// TIA Portal V20 export
// export: Created 2025-12-01T14:57:41.7461211Z, ExportSetting None, DisplayName Totally Integrated Automation Portal, DisplayVersion V20 Update 3, DisplayName TIA Portal Openness, DisplayVersion V20 Update 3, DisplayName TIA Portal Version Control Interface, DisplayVersion V20 Update 3, DisplayName STEP 7 Professional, DisplayVersion V20 Update 3, DisplayName STEP 7 Safety, DisplayVersion V20 Update 2, DisplayName WinCC Basic/Comfort/Advanced, DisplayVersion V20 Update 3, DisplayName WinCC Professional, DisplayVersion V20 Update 3, DisplayName WinCC Unified, DisplayVersion V20 Update 3
FUNCTION_BLOCK "FB381_Transporte_Paletizador_NDD_E12_S23"   // FB381, LAD
TITLE = Control del Ramal de Salidas
{ S7_Optimized_Access := 'FALSE' }
AUTHOR : PASO
NAME : 20160509
VERSION : 3.6
// E1E3_S1S3    (Paletizador NDD)
// stored: AutoNumber false, SetENOAutomatically false
   VAR_INPUT
      Mesa : UInt;   // Mesa de la FB
      Error_Tx : Bool;
      EnTension : Bool;   // Existe Tension en la Mesa
      Termico_Tx : Bool;
      pHsMx_1 : Bool;   // Desactiva si Transferencia controlada
      pHsMx_2 : Bool;   // Desactiva si Transferencia controlada
      pHsMx_PR1 : Bool;   // Si no hay Prot ON
      pHsMx_PR3 : Bool;   // Si no hay Prot ON
      pHsMx_CorteVelo : Bool;
      phsMx_Seguridad : Bool;
      Avance_Tx : Bool;
      Retroceso_Tx : Bool;
      MAnt_DescargaAct_M1 : Bool;
      AVTF_Ent_M1 : Bool;
      P_Mens_Ent_M1 : Bool;
      MAnt_DescargaAct_M3 : Bool;
      AVTF_Ent_M3 : Bool;
      P_Mens_Ent_M3 : Bool;
      PTF_Sal_M1 : Bool;
      FTF_Sal_M1 : Bool;
      PTF_Sal_M3 : Bool;
      FTF_Sal_M3 : Bool;
      Mx_VelocidadLenta_In : Bool;   // Forzar a Velociada Lenta
      F_EnvMens_Mx : Bool;
      OrdSal_S01 : Bool;
      OrdSal_S03 : Bool;
      V_CNT_pHsMx : Int := 300;
      V_CNT_pHsMx_FTF : Int := 50;   // Valor contador para FTF_Mant
      V_CNTSeg_pHsMx : Int := 3000;
      V_CNT_PasoLenta : Int := 3000;
      V_CNT_ApHsMx : Int := 500;
      V_CNTSeg_ApHsMx : Int := 3000;
      V_CNT_pHsMx_E0S0 : Int := 2000;
      V_CNT_Simultaneo : Int := 2000;
      V_InicioSimultaneo : Int := 0;
      V_FinSimultaneo : Int := 0;
      V_TOut_Tx_Mx : Int := 30000;
      V_TMP_Protrusion : Int := 500;
      V_CNT_PerdidapHs : Int := 1000;
   END_VAR
   VAR_OUTPUT
      P_EnvMens_PMx : Bool;
      P_RecepOK_Mx : Bool;
      PTF_Ent_M1 : Bool;
      FTF_Ent_M1 : Bool;
      PTF_Ent_M3 : Bool;
      FTF_Ent_M3 : Bool;
      ATF_Sal_M1 : Bool;
      P_Mens_Sal_M1 : Bool;
      ATF_Sal_M3 : Bool;
      P_Mens_Sal_M3 : Bool;
   END_VAR
   VAR_IN_OUT
      Interlock_TELEV : "NDD_Interlock_TElev";
   END_VAR
   VAR
      Anular_prE1 : Bool;   // ???
      Anular_prS3 : Bool;   // ???
      Mx_ET00 : Bool;
      Mx_ET01 : Bool;
      Mx_ET02 : Bool;
      Mx_ET08 : Bool;
      Mx_ET09 : Bool;
      Mx_ET10 : Bool;
      Mx_ET11 : Bool;
      Mx_ET12 : Bool;
      Mx_ET50 : Bool;
      Mx_ET51 : Bool;
      Mx_ET110 : Bool;
      Mx_ET111 : Bool;
      Mx_ET150 : Bool;
      Mx_ET151 : Bool;
      Mx_ET30 : Bool;
      Mx_ET31 : Bool;
      Mx_ET32 : Bool;
      Mx_ET33 : Bool;
      Mx_ET70 : Bool;
      Mx_ET71 : Bool;
      Mx_ET72 : Bool;
      Selec_M1_Entrada : Bool;
      Selec_M3_Entrada : Bool;
      Selec_M0_Entrada : Bool;
      Selec_M1_Salida : Bool;
      Selec_M3_Salida : Bool;
      Select_M0_Salida : Bool;
      MEnt_DescargaAct : Bool;
      AVTF_MEnt : Bool;
      P_Mens_MEnt : Bool;
      PTF_MEnt : Bool;
      FTF_MEnt : Bool;
      AVTF_MSal : Bool;
      P_Mens_MSal : Bool;
      PTF_MSal : Bool;
      FTF_MSal : Bool;
      FTF_MEnt_M0 : Bool;
      ProtocoloIniciado : Bool;
      CNT_pHsMx_FTF_OK : Bool;
      Simultaneo_Mx : Bool;
      CNT_pHsMx { S7_SetPoint := 'True'} : "FB910_CNT_UHS";
      CNTSeg_pHsMx { S7_SetPoint := 'True'} : "FB910_CNT_UHS";
      CNT_ApHsMx { S7_SetPoint := 'True'} : "FB910_CNT_UHS";
      CNTSeg_ApHsMx { S7_SetPoint := 'True'} : "FB910_CNT_UHS";
      CNT_Simultaneo { S7_SetPoint := 'True'} : "FB910_CNT_UHS";
      CNTEntrada_E0 { S7_SetPoint := 'True'} : "FB910_CNT_UHS";
      CNTSalida_S0 { S7_SetPoint := 'True'} : "FB910_CNT_UHS";
      TMP_EnTension { S7_SetPoint := 'True'} : "FB910_CNT_UHS";
      TOut_Av_Mx { S7_SetPoint := 'True'} : "FB910_CNT_UHS";
      TOut_Ret_Mx { S7_SetPoint := 'True'} : "FB910_CNT_UHS";
      TMP_Protrusion { S7_SetPoint := 'True'} : "FB910_CNT_UHS";
      CNT_PerdidapHs { S7_SetPoint := 'True'} : "FB910_CNT_UHS";
      STAT_EnvMens_PMx : Bool;
   END_VAR
   VAR_TEMP
      EstadoZona : "EstadoZona";
      EstadoVI : "EstadosMesa_Transporte_Paletizador_NDD";
      ConfigFB : "UDT_ConfigFB";   // Configuracion de la FB de la Mesa
      V_Protrusion : Int;
      Aux_ET00 : Bool;
      SinPHS_E0 : Bool;
   END_VAR
   VAR_TEMP   // added for the SCL form of the ladder/FBD networks
      _w1 : Bool;
      _w2 : Bool;
   END_VAR
BEGIN

REGION Network 1: INICIALIZACIONES
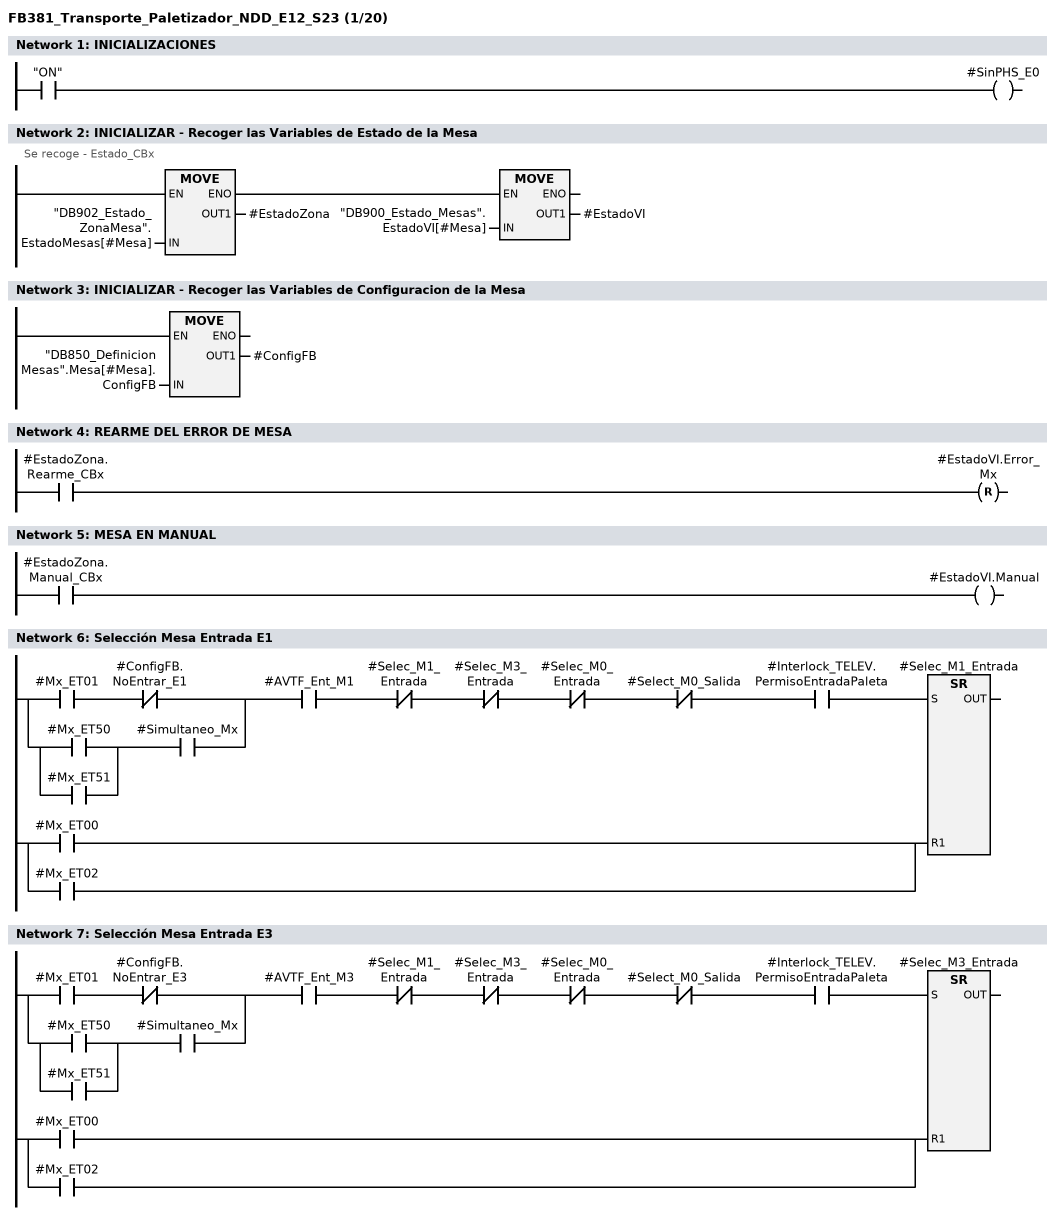
   RUNG wire#powerrail
      Contact( "ON" )
      Coil( #SinPHS_E0 )
   END_RUNG
   // the same network as SCL:
   #SinPHS_E0 := "ON";
END_REGION

REGION Network 2: INICIALIZAR - Recoger las Variables de Estado de la Mesa
   // Se recoge - Estado_CBx
   RUNG wire#powerrail
      Move(in := "DB902_Estado_ZonaMesa".EstadoMesas[#Mesa], out1 => #EstadoZona)
      Move(in := "DB900_Estado_Mesas".EstadoVI[#Mesa], out1 => #EstadoVI)
   END_RUNG
   // the same network as SCL:
   #EstadoZona := "DB902_Estado_ZonaMesa".EstadoMesas[#Mesa];
   #EstadoVI := "DB900_Estado_Mesas".EstadoVI[#Mesa];
END_REGION

REGION Network 3: INICIALIZAR - Recoger las Variables de Configuracion de la Mesa
   RUNG wire#powerrail
      Move(in := "DB850_DefinicionMesas".Mesa[#Mesa].ConfigFB, out1 => #ConfigFB)
   END_RUNG
   // the same network as SCL:
   #ConfigFB := "DB850_DefinicionMesas".Mesa[#Mesa].ConfigFB;
END_REGION

REGION Network 4: REARME DEL ERROR DE MESA
   RUNG wire#powerrail
      Contact( #EstadoZona.Rearme_CBx )
      R_Coil( #EstadoVI.Error_Mx )
   END_RUNG
   // the same network as SCL:
   IF #EstadoZona.Rearme_CBx THEN #EstadoVI.Error_Mx := FALSE; END_IF;
END_REGION

REGION Network 5: MESA EN MANUAL
   RUNG wire#powerrail
      Contact( #EstadoZona.Manual_CBx )
      Coil( #EstadoVI.Manual )
   END_RUNG
   // the same network as SCL:
   #EstadoVI.Manual := #EstadoZona.Manual_CBx;
END_REGION

REGION Network 6: Selección Mesa Entrada E1
   RUNG wire#powerrail
      Contact( #Mx_ET01 )
      I_Contact( #ConfigFB.NoEntrar_E1 )
      wire#w1
      Contact( #AVTF_Ent_M1 )
      I_Contact( #Selec_M1_Entrada )
      I_Contact( #Selec_M3_Entrada )
      I_Contact( #Selec_M0_Entrada )
      I_Contact( #Select_M0_Salida )
      Contact( #Interlock_TELEV.PermisoEntradaPaleta )
      S_SR(operand := #Selec_M1_Entrada, r1 := wire#w3)
   END_RUNG
   RUNG wire#powerrail
      Contact( #Mx_ET50 )
      wire#w2
      Contact( #Simultaneo_Mx )
   END_RUNG wire#w1
   RUNG wire#powerrail
      Contact( #Mx_ET51 )
   END_RUNG wire#w2
   RUNG wire#powerrail
      Contact( #Mx_ET00 )
   END_RUNG wire#w3
   RUNG wire#powerrail
      Contact( #Mx_ET02 )
   END_RUNG wire#w3
   // the same network as SCL:
   IF ((#Mx_ET01 AND NOT #ConfigFB.NoEntrar_E1) OR ((#Mx_ET50 OR #Mx_ET51) AND #Simultaneo_Mx)) AND #AVTF_Ent_M1 AND NOT #Selec_M1_Entrada AND NOT #Selec_M3_Entrada AND NOT #Selec_M0_Entrada AND NOT #Select_M0_Salida AND #Interlock_TELEV.PermisoEntradaPaleta THEN
       #Selec_M1_Entrada := TRUE;   // SR flip-flop
   END_IF;
   IF #Mx_ET00 OR #Mx_ET02 THEN #Selec_M1_Entrada := FALSE; END_IF;
END_REGION

REGION Network 7: Selección Mesa Entrada E3
   RUNG wire#powerrail
      Contact( #Mx_ET01 )
      I_Contact( #ConfigFB.NoEntrar_E3 )
      wire#w1
      Contact( #AVTF_Ent_M3 )
      I_Contact( #Selec_M1_Entrada )
      I_Contact( #Selec_M3_Entrada )
      I_Contact( #Selec_M0_Entrada )
      I_Contact( #Select_M0_Salida )
      Contact( #Interlock_TELEV.PermisoEntradaPaleta )
      S_SR(operand := #Selec_M3_Entrada, r1 := wire#w3)
   END_RUNG
   RUNG wire#powerrail
      Contact( #Mx_ET50 )
      wire#w2
      Contact( #Simultaneo_Mx )
   END_RUNG wire#w1
   RUNG wire#powerrail
      Contact( #Mx_ET51 )
   END_RUNG wire#w2
   RUNG wire#powerrail
      Contact( #Mx_ET00 )
   END_RUNG wire#w3
   RUNG wire#powerrail
      Contact( #Mx_ET02 )
   END_RUNG wire#w3
   // the same network as SCL:
   IF ((#Mx_ET01 AND NOT #ConfigFB.NoEntrar_E3) OR ((#Mx_ET50 OR #Mx_ET51) AND #Simultaneo_Mx)) AND #AVTF_Ent_M3 AND NOT #Selec_M1_Entrada AND NOT #Selec_M3_Entrada AND NOT #Selec_M0_Entrada AND NOT #Select_M0_Salida AND #Interlock_TELEV.PermisoEntradaPaleta THEN
       #Selec_M3_Entrada := TRUE;   // SR flip-flop
   END_IF;
   IF #Mx_ET00 OR #Mx_ET02 THEN #Selec_M3_Entrada := FALSE; END_IF;
END_REGION

REGION Network 8: Selección Mesa Salida S1
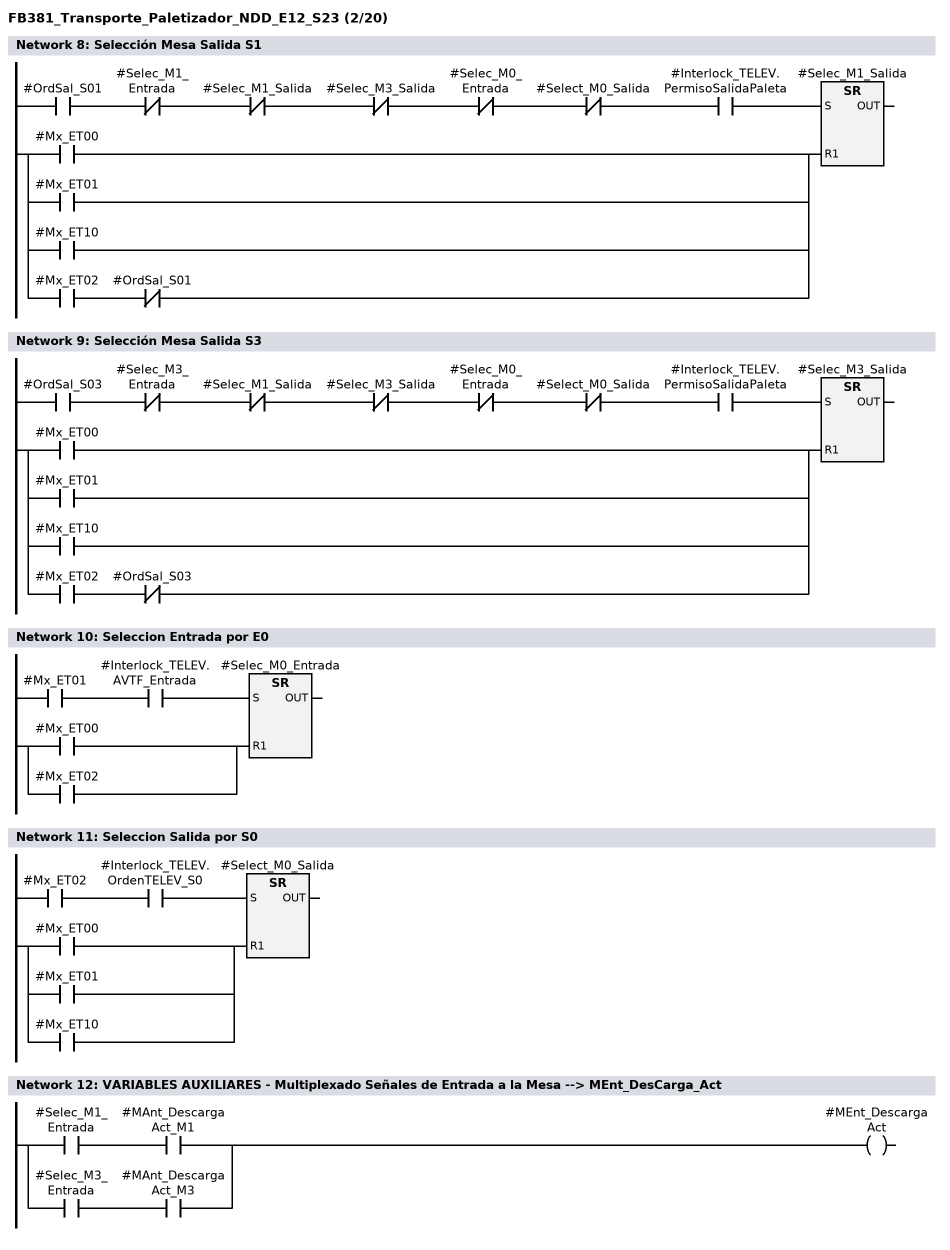
   RUNG wire#powerrail
      Contact( #OrdSal_S01 )
      I_Contact( #Selec_M1_Entrada )
      I_Contact( #Selec_M1_Salida )
      I_Contact( #Selec_M3_Salida )
      I_Contact( #Selec_M0_Entrada )
      I_Contact( #Select_M0_Salida )
      Contact( #Interlock_TELEV.PermisoSalidaPaleta )
      S_SR(operand := #Selec_M1_Salida, r1 := wire#w1)
   END_RUNG
   RUNG wire#powerrail
      Contact( #Mx_ET00 )
   END_RUNG wire#w1
   RUNG wire#powerrail
      Contact( #Mx_ET01 )
   END_RUNG wire#w1
   RUNG wire#powerrail
      Contact( #Mx_ET10 )
   END_RUNG wire#w1
   RUNG wire#powerrail
      Contact( #Mx_ET02 )
      I_Contact( #OrdSal_S01 )
   END_RUNG wire#w1
   // the same network as SCL:
   IF #OrdSal_S01 AND NOT #Selec_M1_Entrada AND NOT #Selec_M1_Salida AND NOT #Selec_M3_Salida AND NOT #Selec_M0_Entrada AND NOT #Select_M0_Salida AND #Interlock_TELEV.PermisoSalidaPaleta THEN
       #Selec_M1_Salida := TRUE;   // SR flip-flop
   END_IF;
   IF #Mx_ET00 OR #Mx_ET01 OR #Mx_ET10 OR (#Mx_ET02 AND NOT #OrdSal_S01) THEN
       #Selec_M1_Salida := FALSE;
   END_IF;
END_REGION

REGION Network 9: Selección Mesa Salida S3
   RUNG wire#powerrail
      Contact( #OrdSal_S03 )
      I_Contact( #Selec_M3_Entrada )
      I_Contact( #Selec_M1_Salida )
      I_Contact( #Selec_M3_Salida )
      I_Contact( #Selec_M0_Entrada )
      I_Contact( #Select_M0_Salida )
      Contact( #Interlock_TELEV.PermisoSalidaPaleta )
      S_SR(operand := #Selec_M3_Salida, r1 := wire#w1)
   END_RUNG
   RUNG wire#powerrail
      Contact( #Mx_ET00 )
   END_RUNG wire#w1
   RUNG wire#powerrail
      Contact( #Mx_ET01 )
   END_RUNG wire#w1
   RUNG wire#powerrail
      Contact( #Mx_ET10 )
   END_RUNG wire#w1
   RUNG wire#powerrail
      Contact( #Mx_ET02 )
      I_Contact( #OrdSal_S03 )
   END_RUNG wire#w1
   // the same network as SCL:
   IF #OrdSal_S03 AND NOT #Selec_M3_Entrada AND NOT #Selec_M1_Salida AND NOT #Selec_M3_Salida AND NOT #Selec_M0_Entrada AND NOT #Select_M0_Salida AND #Interlock_TELEV.PermisoSalidaPaleta THEN
       #Selec_M3_Salida := TRUE;   // SR flip-flop
   END_IF;
   IF #Mx_ET00 OR #Mx_ET01 OR #Mx_ET10 OR (#Mx_ET02 AND NOT #OrdSal_S03) THEN
       #Selec_M3_Salida := FALSE;
   END_IF;
END_REGION

REGION Network 10: Seleccion Entrada por E0
   RUNG wire#powerrail
      Contact( #Mx_ET01 )
      Contact( #Interlock_TELEV.AVTF_Entrada )
      S_SR(operand := #Selec_M0_Entrada, r1 := wire#w1)
   END_RUNG
   RUNG wire#powerrail
      Contact( #Mx_ET00 )
   END_RUNG wire#w1
   RUNG wire#powerrail
      Contact( #Mx_ET02 )
   END_RUNG wire#w1
   // the same network as SCL:
   IF #Mx_ET01 AND #Interlock_TELEV.AVTF_Entrada THEN
       #Selec_M0_Entrada := TRUE;   // SR flip-flop
   END_IF;
   IF #Mx_ET00 OR #Mx_ET02 THEN #Selec_M0_Entrada := FALSE; END_IF;
END_REGION

REGION Network 11: Seleccion Salida por S0
   RUNG wire#powerrail
      Contact( #Mx_ET02 )
      Contact( #Interlock_TELEV.OrdenTELEV_S0 )
      S_SR(operand := #Select_M0_Salida, r1 := wire#w1)
   END_RUNG
   RUNG wire#powerrail
      Contact( #Mx_ET00 )
   END_RUNG wire#w1
   RUNG wire#powerrail
      Contact( #Mx_ET01 )
   END_RUNG wire#w1
   RUNG wire#powerrail
      Contact( #Mx_ET10 )
   END_RUNG wire#w1
   // the same network as SCL:
   IF #Mx_ET02 AND #Interlock_TELEV.OrdenTELEV_S0 THEN
       #Select_M0_Salida := TRUE;   // SR flip-flop
   END_IF;
   IF #Mx_ET00 OR #Mx_ET01 OR #Mx_ET10 THEN #Select_M0_Salida := FALSE; END_IF;
END_REGION

REGION Network 12: VARIABLES AUXILIARES - Multiplexado Señales de Entrada a la Mesa --> MEnt_DesCarga_Act
   RUNG wire#powerrail
      Contact( #Selec_M1_Entrada )
      Contact( #MAnt_DescargaAct_M1 )
      wire#w1
      Coil( #MEnt_DescargaAct )
   END_RUNG
   RUNG wire#powerrail
      Contact( #Selec_M3_Entrada )
      Contact( #MAnt_DescargaAct_M3 )
   END_RUNG wire#w1
   // the same network as SCL:
   #MEnt_DescargaAct := (#Selec_M1_Entrada AND #MAnt_DescargaAct_M1) OR (#Selec_M3_Entrada AND #MAnt_DescargaAct_M3);
END_REGION

REGION Network 13: VARIABLES AUXILIARES - Multiplexado Señales de Entrada a la Mesa --> AVTF_MEnt
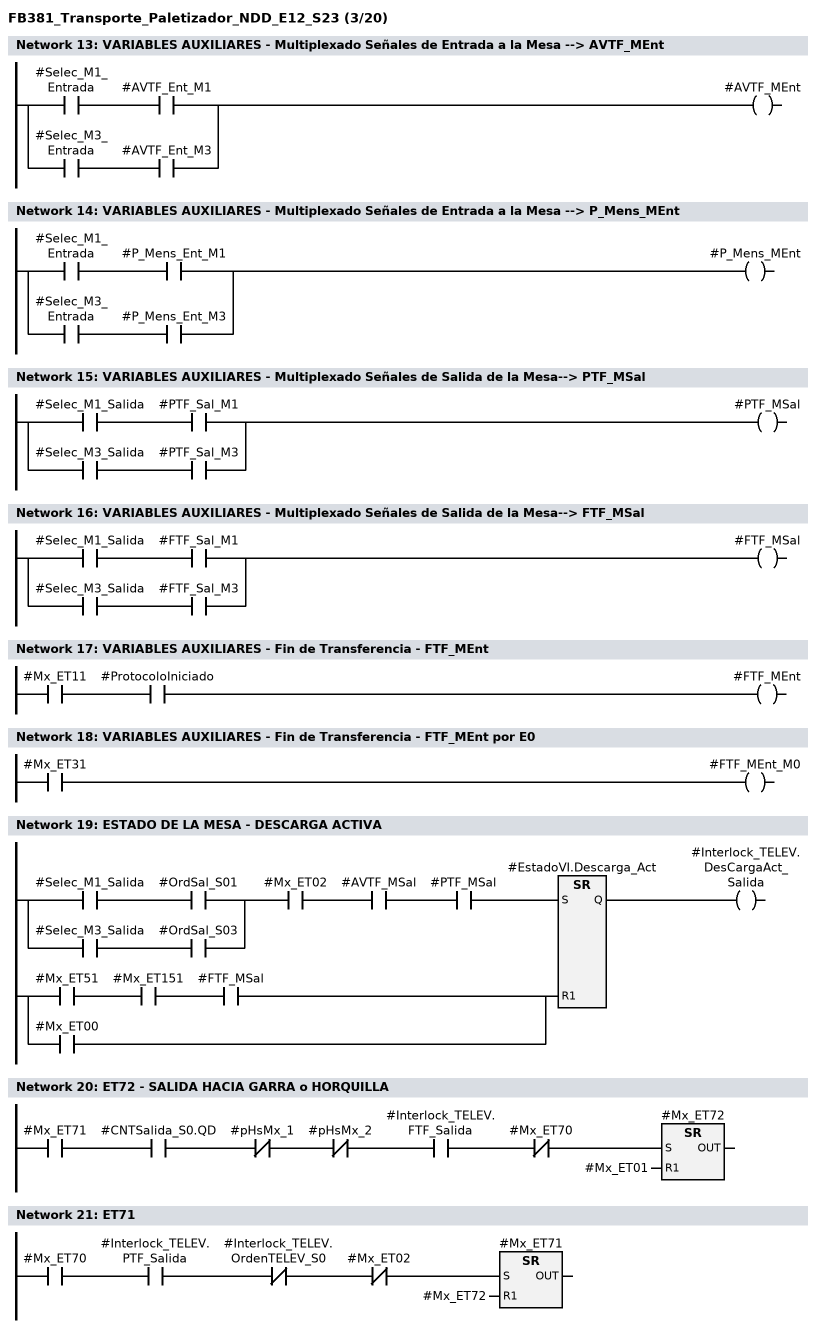
   RUNG wire#powerrail
      Contact( #Selec_M1_Entrada )
      Contact( #AVTF_Ent_M1 )
      wire#w1
      Coil( #AVTF_MEnt )
   END_RUNG
   RUNG wire#powerrail
      Contact( #Selec_M3_Entrada )
      Contact( #AVTF_Ent_M3 )
   END_RUNG wire#w1
   // the same network as SCL:
   #AVTF_MEnt := (#Selec_M1_Entrada AND #AVTF_Ent_M1) OR (#Selec_M3_Entrada AND #AVTF_Ent_M3);
END_REGION

REGION Network 14: VARIABLES AUXILIARES - Multiplexado Señales de Entrada a la Mesa --> P_Mens_MEnt
   RUNG wire#powerrail
      Contact( #Selec_M1_Entrada )
      Contact( #P_Mens_Ent_M1 )
      wire#w1
      Coil( #P_Mens_MEnt )
   END_RUNG
   RUNG wire#powerrail
      Contact( #Selec_M3_Entrada )
      Contact( #P_Mens_Ent_M3 )
   END_RUNG wire#w1
   // the same network as SCL:
   #P_Mens_MEnt := (#Selec_M1_Entrada AND #P_Mens_Ent_M1) OR (#Selec_M3_Entrada AND #P_Mens_Ent_M3);
END_REGION

REGION Network 15: VARIABLES AUXILIARES - Multiplexado Señales de Salida de la Mesa--> PTF_MSal
   RUNG wire#powerrail
      Contact( #Selec_M1_Salida )
      Contact( #PTF_Sal_M1 )
      wire#w1
      Coil( #PTF_MSal )
   END_RUNG
   RUNG wire#powerrail
      Contact( #Selec_M3_Salida )
      Contact( #PTF_Sal_M3 )
   END_RUNG wire#w1
   // the same network as SCL:
   #PTF_MSal := (#Selec_M1_Salida AND #PTF_Sal_M1) OR (#Selec_M3_Salida AND #PTF_Sal_M3);
END_REGION

REGION Network 16: VARIABLES AUXILIARES - Multiplexado Señales de Salida de la Mesa--> FTF_MSal
   RUNG wire#powerrail
      Contact( #Selec_M1_Salida )
      Contact( #FTF_Sal_M1 )
      wire#w1
      Coil( #FTF_MSal )
   END_RUNG
   RUNG wire#powerrail
      Contact( #Selec_M3_Salida )
      Contact( #FTF_Sal_M3 )
   END_RUNG wire#w1
   // the same network as SCL:
   #FTF_MSal := (#Selec_M1_Salida AND #FTF_Sal_M1) OR (#Selec_M3_Salida AND #FTF_Sal_M3);
END_REGION

REGION Network 17: VARIABLES AUXILIARES - Fin de Transferencia - FTF_MEnt
   RUNG wire#powerrail
      Contact( #Mx_ET11 )
      Contact( #ProtocoloIniciado )
      Coil( #FTF_MEnt )
   END_RUNG
   // the same network as SCL:
   #FTF_MEnt := #Mx_ET11 AND #ProtocoloIniciado;
END_REGION

REGION Network 18: VARIABLES AUXILIARES - Fin de Transferencia - FTF_MEnt por E0
   RUNG wire#powerrail
      Contact( #Mx_ET31 )
      Coil( #FTF_MEnt_M0 )
   END_RUNG
   // the same network as SCL:
   #FTF_MEnt_M0 := #Mx_ET31;
END_REGION

REGION Network 19: ESTADO DE LA MESA - DESCARGA ACTIVA
   RUNG wire#powerrail
      Contact( #Selec_M1_Salida )
      Contact( #OrdSal_S01 )
      wire#w1
      Contact( #Mx_ET02 )
      Contact( #AVTF_MSal )
      Contact( #PTF_MSal )
      S_SR(operand := #EstadoVI.Descarga_Act, r1 := wire#w2)
      Coil( #Interlock_TELEV.DesCargaAct_Salida )
   END_RUNG
   RUNG wire#powerrail
      Contact( #Selec_M3_Salida )
      Contact( #OrdSal_S03 )
   END_RUNG wire#w1
   RUNG wire#powerrail
      Contact( #Mx_ET51 )
      Contact( #Mx_ET151 )
      Contact( #FTF_MSal )
   END_RUNG wire#w2
   RUNG wire#powerrail
      Contact( #Mx_ET00 )
   END_RUNG wire#w2
   // the same network as SCL:
   IF ((#Selec_M1_Salida AND #OrdSal_S01) OR (#Selec_M3_Salida AND #OrdSal_S03)) AND #Mx_ET02 AND #AVTF_MSal AND #PTF_MSal THEN
       #EstadoVI.Descarga_Act := TRUE;   // SR flip-flop
   END_IF;
   IF (#Mx_ET51 AND #Mx_ET151 AND #FTF_MSal) OR #Mx_ET00 THEN #EstadoVI.Descarga_Act := FALSE; END_IF;
   #Interlock_TELEV.DesCargaAct_Salida := #EstadoVI.Descarga_Act;
END_REGION

REGION Network 20: ET72 - SALIDA HACIA GARRA o HORQUILLA
   RUNG wire#powerrail
      Contact( #Mx_ET71 )
      Contact( #CNTSalida_S0.QD )
      I_Contact( #pHsMx_1 )
      I_Contact( #pHsMx_2 )
      Contact( #Interlock_TELEV.FTF_Salida )
      I_Contact( #Mx_ET70 )
      S_SR(operand := #Mx_ET72, r1 := #Mx_ET01)
   END_RUNG
   // the same network as SCL:
   IF #Mx_ET71 AND #CNTSalida_S0.QD AND NOT #pHsMx_1 AND NOT #pHsMx_2 AND #Interlock_TELEV.FTF_Salida AND NOT #Mx_ET70 THEN
       #Mx_ET72 := TRUE;   // SR flip-flop
   END_IF;
   IF #Mx_ET01 THEN #Mx_ET72 := FALSE; END_IF;
END_REGION

REGION Network 21: ET71
   RUNG wire#powerrail
      Contact( #Mx_ET70 )
      Contact( #Interlock_TELEV.PTF_Salida )
      I_Contact( #Interlock_TELEV.OrdenTELEV_S0 )
      I_Contact( #Mx_ET02 )
      S_SR(operand := #Mx_ET71, r1 := #Mx_ET72)
   END_RUNG
   // the same network as SCL:
   IF #Mx_ET70 AND #Interlock_TELEV.PTF_Salida AND NOT #Interlock_TELEV.OrdenTELEV_S0 AND NOT #Mx_ET02 THEN
       #Mx_ET71 := TRUE;   // SR flip-flop
   END_IF;
   IF #Mx_ET72 THEN #Mx_ET71 := FALSE; END_IF;
END_REGION

REGION Network 22: ET70
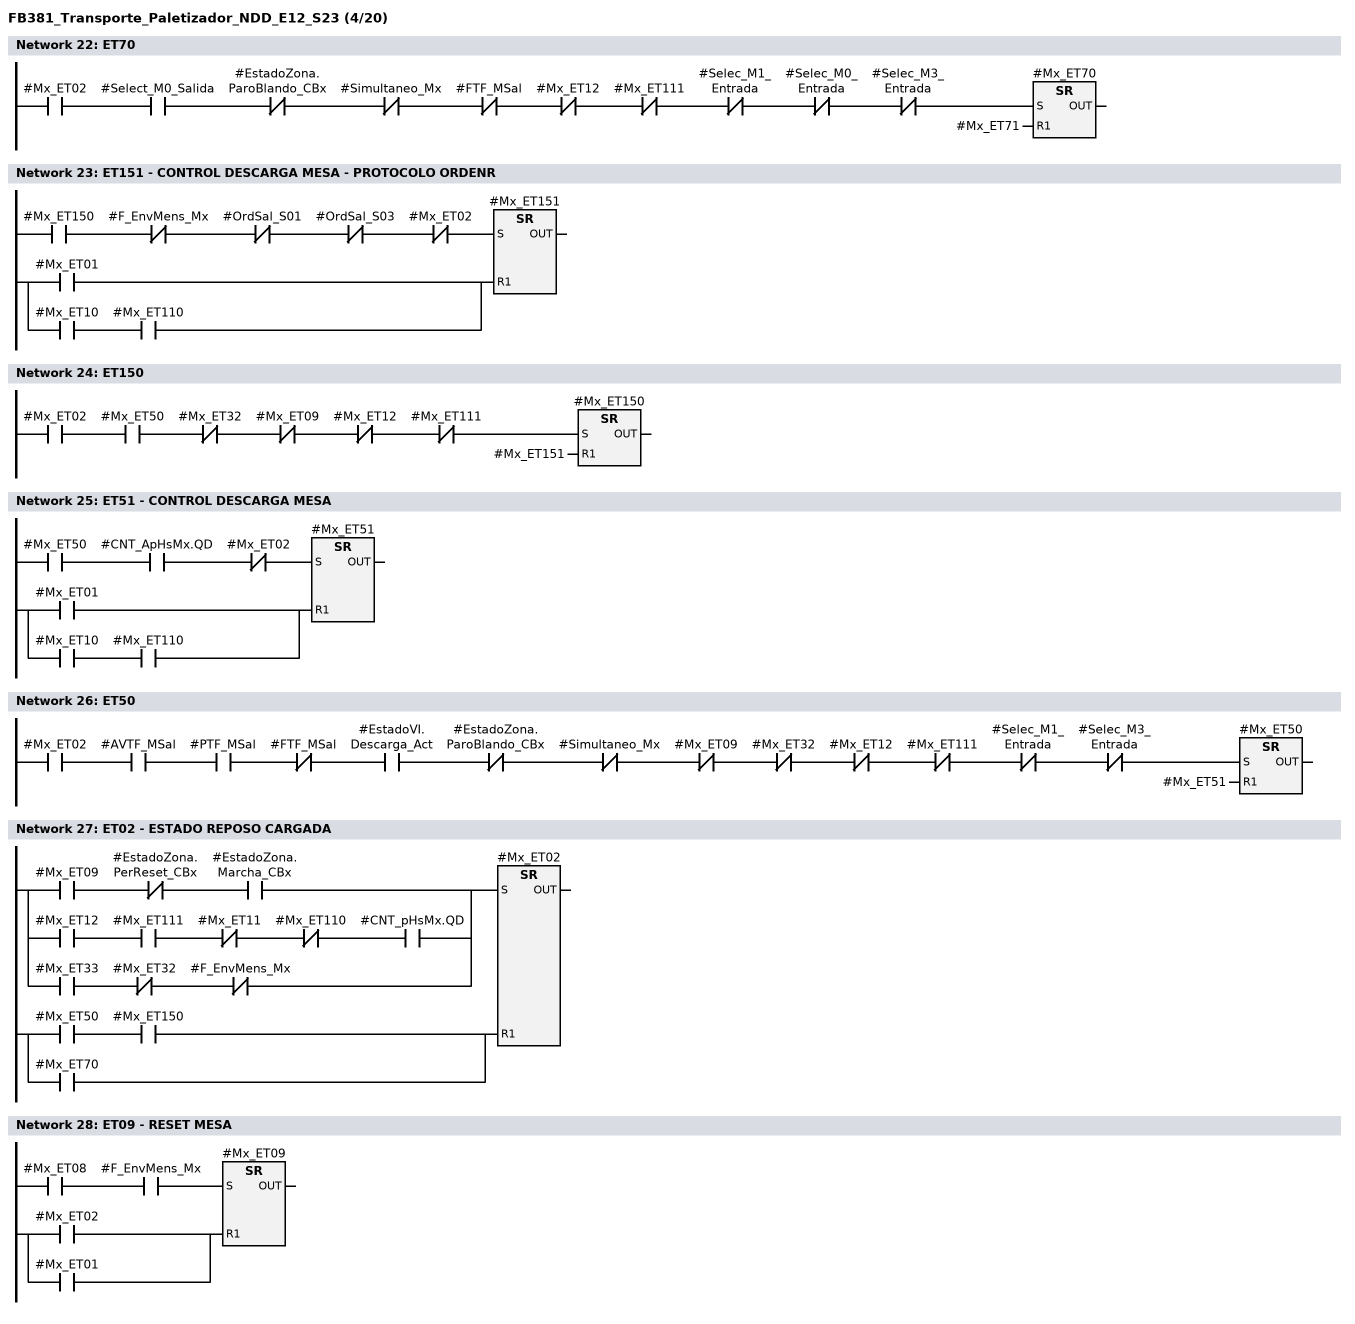
   RUNG wire#powerrail
      Contact( #Mx_ET02 )
      Contact( #Select_M0_Salida )
      I_Contact( #EstadoZona.ParoBlando_CBx )
      I_Contact( #Simultaneo_Mx )
      I_Contact( #FTF_MSal )
      I_Contact( #Mx_ET12 )
      I_Contact( #Mx_ET111 )
      I_Contact( #Selec_M1_Entrada )
      I_Contact( #Selec_M0_Entrada )
      I_Contact( #Selec_M3_Entrada )
      S_SR(operand := #Mx_ET70, r1 := #Mx_ET71)
   END_RUNG
   // the same network as SCL:
   IF #Mx_ET02 AND #Select_M0_Salida AND NOT #EstadoZona.ParoBlando_CBx AND NOT #Simultaneo_Mx AND NOT #FTF_MSal AND NOT #Mx_ET12 AND NOT #Mx_ET111 AND NOT #Selec_M1_Entrada AND NOT #Selec_M0_Entrada AND NOT #Selec_M3_Entrada THEN
       #Mx_ET70 := TRUE;   // SR flip-flop
   END_IF;
   IF #Mx_ET71 THEN #Mx_ET70 := FALSE; END_IF;
END_REGION

REGION Network 23: ET151 - CONTROL DESCARGA MESA - PROTOCOLO ORDENR
   RUNG wire#powerrail
      Contact( #Mx_ET150 )
      I_Contact( #F_EnvMens_Mx )
      I_Contact( #OrdSal_S01 )
      I_Contact( #OrdSal_S03 )
      I_Contact( #Mx_ET02 )
      S_SR(operand := #Mx_ET151, r1 := wire#w1)
   END_RUNG
   RUNG wire#powerrail
      Contact( #Mx_ET01 )
   END_RUNG wire#w1
   RUNG wire#powerrail
      Contact( #Mx_ET10 )
      Contact( #Mx_ET110 )
   END_RUNG wire#w1
   // the same network as SCL:
   IF #Mx_ET150 AND NOT #F_EnvMens_Mx AND NOT #OrdSal_S01 AND NOT #OrdSal_S03 AND NOT #Mx_ET02 THEN
       #Mx_ET151 := TRUE;   // SR flip-flop
   END_IF;
   IF #Mx_ET01 OR (#Mx_ET10 AND #Mx_ET110) THEN #Mx_ET151 := FALSE; END_IF;
END_REGION

REGION Network 24: ET150
   RUNG wire#powerrail
      Contact( #Mx_ET02 )
      Contact( #Mx_ET50 )
      I_Contact( #Mx_ET32 )
      I_Contact( #Mx_ET09 )
      I_Contact( #Mx_ET12 )
      I_Contact( #Mx_ET111 )
      S_SR(operand := #Mx_ET150, r1 := #Mx_ET151)
   END_RUNG
   // the same network as SCL:
   IF #Mx_ET02 AND #Mx_ET50 AND NOT #Mx_ET32 AND NOT #Mx_ET09 AND NOT #Mx_ET12 AND NOT #Mx_ET111 THEN
       #Mx_ET150 := TRUE;   // SR flip-flop
   END_IF;
   IF #Mx_ET151 THEN #Mx_ET150 := FALSE; END_IF;
END_REGION

REGION Network 25: ET51 - CONTROL DESCARGA MESA
   RUNG wire#powerrail
      Contact( #Mx_ET50 )
      Contact( #CNT_ApHsMx.QD )
      I_Contact( #Mx_ET02 )
      S_SR(operand := #Mx_ET51, r1 := wire#w1)
   END_RUNG
   RUNG wire#powerrail
      Contact( #Mx_ET01 )
   END_RUNG wire#w1
   RUNG wire#powerrail
      Contact( #Mx_ET10 )
      Contact( #Mx_ET110 )
   END_RUNG wire#w1
   // the same network as SCL:
   IF #Mx_ET50 AND #CNT_ApHsMx.QD AND NOT #Mx_ET02 THEN
       #Mx_ET51 := TRUE;   // SR flip-flop
   END_IF;
   IF #Mx_ET01 OR (#Mx_ET10 AND #Mx_ET110) THEN #Mx_ET51 := FALSE; END_IF;
END_REGION

REGION Network 26: ET50
   RUNG wire#powerrail
      Contact( #Mx_ET02 )
      Contact( #AVTF_MSal )
      Contact( #PTF_MSal )
      I_Contact( #FTF_MSal )
      Contact( #EstadoVI.Descarga_Act )
      I_Contact( #EstadoZona.ParoBlando_CBx )
      I_Contact( #Simultaneo_Mx )
      I_Contact( #Mx_ET09 )
      I_Contact( #Mx_ET32 )
      I_Contact( #Mx_ET12 )
      I_Contact( #Mx_ET111 )
      I_Contact( #Selec_M1_Entrada )
      I_Contact( #Selec_M3_Entrada )
      S_SR(operand := #Mx_ET50, r1 := #Mx_ET51)
   END_RUNG
   // the same network as SCL:
   IF #Mx_ET02 AND #AVTF_MSal AND #PTF_MSal AND NOT #FTF_MSal AND #EstadoVI.Descarga_Act AND NOT #EstadoZona.ParoBlando_CBx AND NOT #Simultaneo_Mx AND NOT #Mx_ET09 AND NOT #Mx_ET32 AND NOT #Mx_ET12 AND NOT #Mx_ET111 AND NOT #Selec_M1_Entrada AND NOT #Selec_M3_Entrada THEN
       #Mx_ET50 := TRUE;   // SR flip-flop
   END_IF;
   IF #Mx_ET51 THEN #Mx_ET50 := FALSE; END_IF;
END_REGION

REGION Network 27: ET02 - ESTADO REPOSO CARGADA
   RUNG wire#powerrail
      Contact( #Mx_ET09 )
      I_Contact( #EstadoZona.PerReset_CBx )
      Contact( #EstadoZona.Marcha_CBx )
      wire#w1
      S_SR(operand := #Mx_ET02, r1 := wire#w2)
   END_RUNG
   RUNG wire#powerrail
      Contact( #Mx_ET12 )
      Contact( #Mx_ET111 )
      I_Contact( #Mx_ET11 )
      I_Contact( #Mx_ET110 )
      Contact( #CNT_pHsMx.QD )
   END_RUNG wire#w1
   RUNG wire#powerrail
      Contact( #Mx_ET33 )
      I_Contact( #Mx_ET32 )
      I_Contact( #F_EnvMens_Mx )
   END_RUNG wire#w1
   RUNG wire#powerrail
      Contact( #Mx_ET50 )
      Contact( #Mx_ET150 )
   END_RUNG wire#w2
   RUNG wire#powerrail
      Contact( #Mx_ET70 )
   END_RUNG wire#w2
   // the same network as SCL:
   IF (#Mx_ET09 AND NOT #EstadoZona.PerReset_CBx AND #EstadoZona.Marcha_CBx) OR (#Mx_ET12 AND #Mx_ET111 AND NOT #Mx_ET11 AND NOT #Mx_ET110 AND #CNT_pHsMx.QD) OR (#Mx_ET33 AND NOT #Mx_ET32 AND NOT #F_EnvMens_Mx) THEN
       #Mx_ET02 := TRUE;   // SR flip-flop
   END_IF;
   IF (#Mx_ET50 AND #Mx_ET150) OR #Mx_ET70 THEN #Mx_ET02 := FALSE; END_IF;
END_REGION

REGION Network 28: ET09 - RESET MESA
   RUNG wire#powerrail
      Contact( #Mx_ET08 )
      Contact( #F_EnvMens_Mx )
      S_SR(operand := #Mx_ET09, r1 := wire#w1)
   END_RUNG
   RUNG wire#powerrail
      Contact( #Mx_ET02 )
   END_RUNG wire#w1
   RUNG wire#powerrail
      Contact( #Mx_ET01 )
   END_RUNG wire#w1
   // the same network as SCL:
   IF #Mx_ET08 AND #F_EnvMens_Mx THEN
       #Mx_ET09 := TRUE;   // SR flip-flop
   END_IF;
   IF #Mx_ET02 OR #Mx_ET01 THEN #Mx_ET09 := FALSE; END_IF;
END_REGION

REGION Network 29: ET08
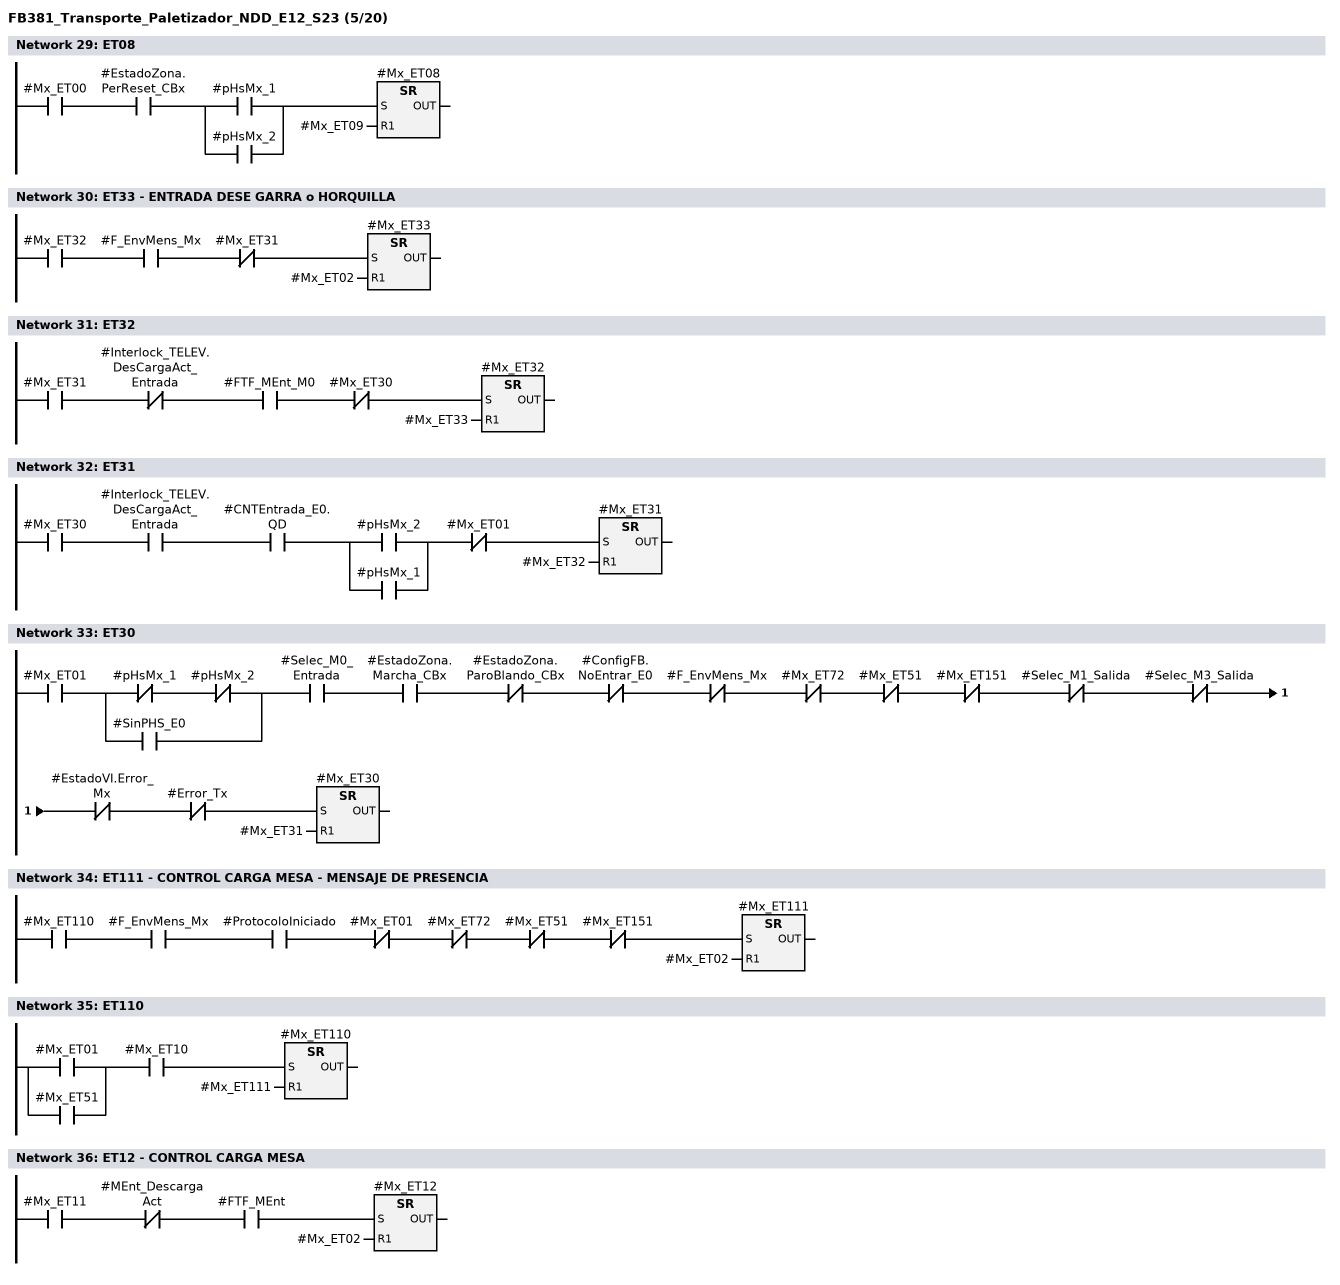
   RUNG wire#powerrail
      Contact( #Mx_ET00 )
      Contact( #EstadoZona.PerReset_CBx )
      wire#w1
      Contact( #pHsMx_1 )
      wire#w2
      S_SR(operand := #Mx_ET08, r1 := #Mx_ET09)
   END_RUNG
   RUNG wire#w1
      Contact( #pHsMx_2 )
   END_RUNG wire#w2
   // the same network as SCL:
   IF #Mx_ET00 AND #EstadoZona.PerReset_CBx AND (#pHsMx_1 OR #pHsMx_2) THEN
       #Mx_ET08 := TRUE;   // SR flip-flop
   END_IF;
   IF #Mx_ET09 THEN #Mx_ET08 := FALSE; END_IF;
END_REGION

REGION Network 30: ET33 - ENTRADA DESE GARRA o HORQUILLA
   RUNG wire#powerrail
      Contact( #Mx_ET32 )
      Contact( #F_EnvMens_Mx )
      I_Contact( #Mx_ET31 )
      S_SR(operand := #Mx_ET33, r1 := #Mx_ET02)
   END_RUNG
   // the same network as SCL:
   IF #Mx_ET32 AND #F_EnvMens_Mx AND NOT #Mx_ET31 THEN
       #Mx_ET33 := TRUE;   // SR flip-flop
   END_IF;
   IF #Mx_ET02 THEN #Mx_ET33 := FALSE; END_IF;
END_REGION

REGION Network 31: ET32
   RUNG wire#powerrail
      Contact( #Mx_ET31 )
      I_Contact( #Interlock_TELEV.DesCargaAct_Entrada )
      Contact( #FTF_MEnt_M0 )
      I_Contact( #Mx_ET30 )
      S_SR(operand := #Mx_ET32, r1 := #Mx_ET33)
   END_RUNG
   // the same network as SCL:
   IF #Mx_ET31 AND NOT #Interlock_TELEV.DesCargaAct_Entrada AND #FTF_MEnt_M0 AND NOT #Mx_ET30 THEN
       #Mx_ET32 := TRUE;   // SR flip-flop
   END_IF;
   IF #Mx_ET33 THEN #Mx_ET32 := FALSE; END_IF;
END_REGION

REGION Network 32: ET31
   RUNG wire#powerrail
      Contact( #Mx_ET30 )
      Contact( #Interlock_TELEV.DesCargaAct_Entrada )
      Contact( #CNTEntrada_E0.QD )
      wire#w1
      Contact( #pHsMx_2 )
      wire#w2
      I_Contact( #Mx_ET01 )
      S_SR(operand := #Mx_ET31, r1 := #Mx_ET32)
   END_RUNG
   RUNG wire#w1
      Contact( #pHsMx_1 )
   END_RUNG wire#w2
   // the same network as SCL:
   IF #Mx_ET30 AND #Interlock_TELEV.DesCargaAct_Entrada AND #CNTEntrada_E0.QD AND (#pHsMx_2 OR #pHsMx_1) AND NOT #Mx_ET01 THEN
       #Mx_ET31 := TRUE;   // SR flip-flop
   END_IF;
   IF #Mx_ET32 THEN #Mx_ET31 := FALSE; END_IF;
END_REGION

REGION Network 33: ET30
   RUNG wire#powerrail
      Contact( #Mx_ET01 )
      wire#w1
      I_Contact( #pHsMx_1 )
      I_Contact( #pHsMx_2 )
      wire#w2
      Contact( #Selec_M0_Entrada )
      Contact( #EstadoZona.Marcha_CBx )
      I_Contact( #EstadoZona.ParoBlando_CBx )
      I_Contact( #ConfigFB.NoEntrar_E0 )
      I_Contact( #F_EnvMens_Mx )
      I_Contact( #Mx_ET72 )
      I_Contact( #Mx_ET51 )
      I_Contact( #Mx_ET151 )
      I_Contact( #Selec_M1_Salida )
      I_Contact( #Selec_M3_Salida )
      I_Contact( #EstadoVI.Error_Mx )
      I_Contact( #Error_Tx )
      S_SR(operand := #Mx_ET30, r1 := #Mx_ET31)
   END_RUNG
   RUNG wire#w1
      Contact( #SinPHS_E0 )
   END_RUNG wire#w2
   // the same network as SCL:
   IF #Mx_ET01 AND ((NOT #pHsMx_1 AND NOT #pHsMx_2) OR #SinPHS_E0) AND #Selec_M0_Entrada AND #EstadoZona.Marcha_CBx AND NOT #EstadoZona.ParoBlando_CBx AND NOT #ConfigFB.NoEntrar_E0 AND NOT #F_EnvMens_Mx AND NOT #Mx_ET72 AND NOT #Mx_ET51 AND NOT #Mx_ET151 AND NOT #Selec_M1_Salida AND NOT #Selec_M3_Salida AND NOT #EstadoVI.Error_Mx AND NOT #Error_Tx THEN
       #Mx_ET30 := TRUE;   // SR flip-flop
   END_IF;
   IF #Mx_ET31 THEN #Mx_ET30 := FALSE; END_IF;
END_REGION

REGION Network 34: ET111 - CONTROL CARGA MESA - MENSAJE DE PRESENCIA
   RUNG wire#powerrail
      Contact( #Mx_ET110 )
      Contact( #F_EnvMens_Mx )
      Contact( #ProtocoloIniciado )
      I_Contact( #Mx_ET01 )
      I_Contact( #Mx_ET72 )
      I_Contact( #Mx_ET51 )
      I_Contact( #Mx_ET151 )
      S_SR(operand := #Mx_ET111, r1 := #Mx_ET02)
   END_RUNG
   // the same network as SCL:
   IF #Mx_ET110 AND #F_EnvMens_Mx AND #ProtocoloIniciado AND NOT #Mx_ET01 AND NOT #Mx_ET72 AND NOT #Mx_ET51 AND NOT #Mx_ET151 THEN
       #Mx_ET111 := TRUE;   // SR flip-flop
   END_IF;
   IF #Mx_ET02 THEN #Mx_ET111 := FALSE; END_IF;
END_REGION

REGION Network 35: ET110
   RUNG wire#powerrail
      Contact( #Mx_ET01 )
      wire#w1
      Contact( #Mx_ET10 )
      S_SR(operand := #Mx_ET110, r1 := #Mx_ET111)
   END_RUNG
   RUNG wire#powerrail
      Contact( #Mx_ET51 )
   END_RUNG wire#w1
   // the same network as SCL:
   IF (#Mx_ET01 OR #Mx_ET51) AND #Mx_ET10 THEN
       #Mx_ET110 := TRUE;   // SR flip-flop
   END_IF;
   IF #Mx_ET111 THEN #Mx_ET110 := FALSE; END_IF;
END_REGION

REGION Network 36: ET12 - CONTROL CARGA MESA
   RUNG wire#powerrail
      Contact( #Mx_ET11 )
      I_Contact( #MEnt_DescargaAct )
      Contact( #FTF_MEnt )
      S_SR(operand := #Mx_ET12, r1 := #Mx_ET02)
   END_RUNG
   // the same network as SCL:
   IF #Mx_ET11 AND NOT #MEnt_DescargaAct AND #FTF_MEnt THEN
       #Mx_ET12 := TRUE;   // SR flip-flop
   END_IF;
   IF #Mx_ET02 THEN #Mx_ET12 := FALSE; END_IF;
END_REGION

REGION Network 37: ET11
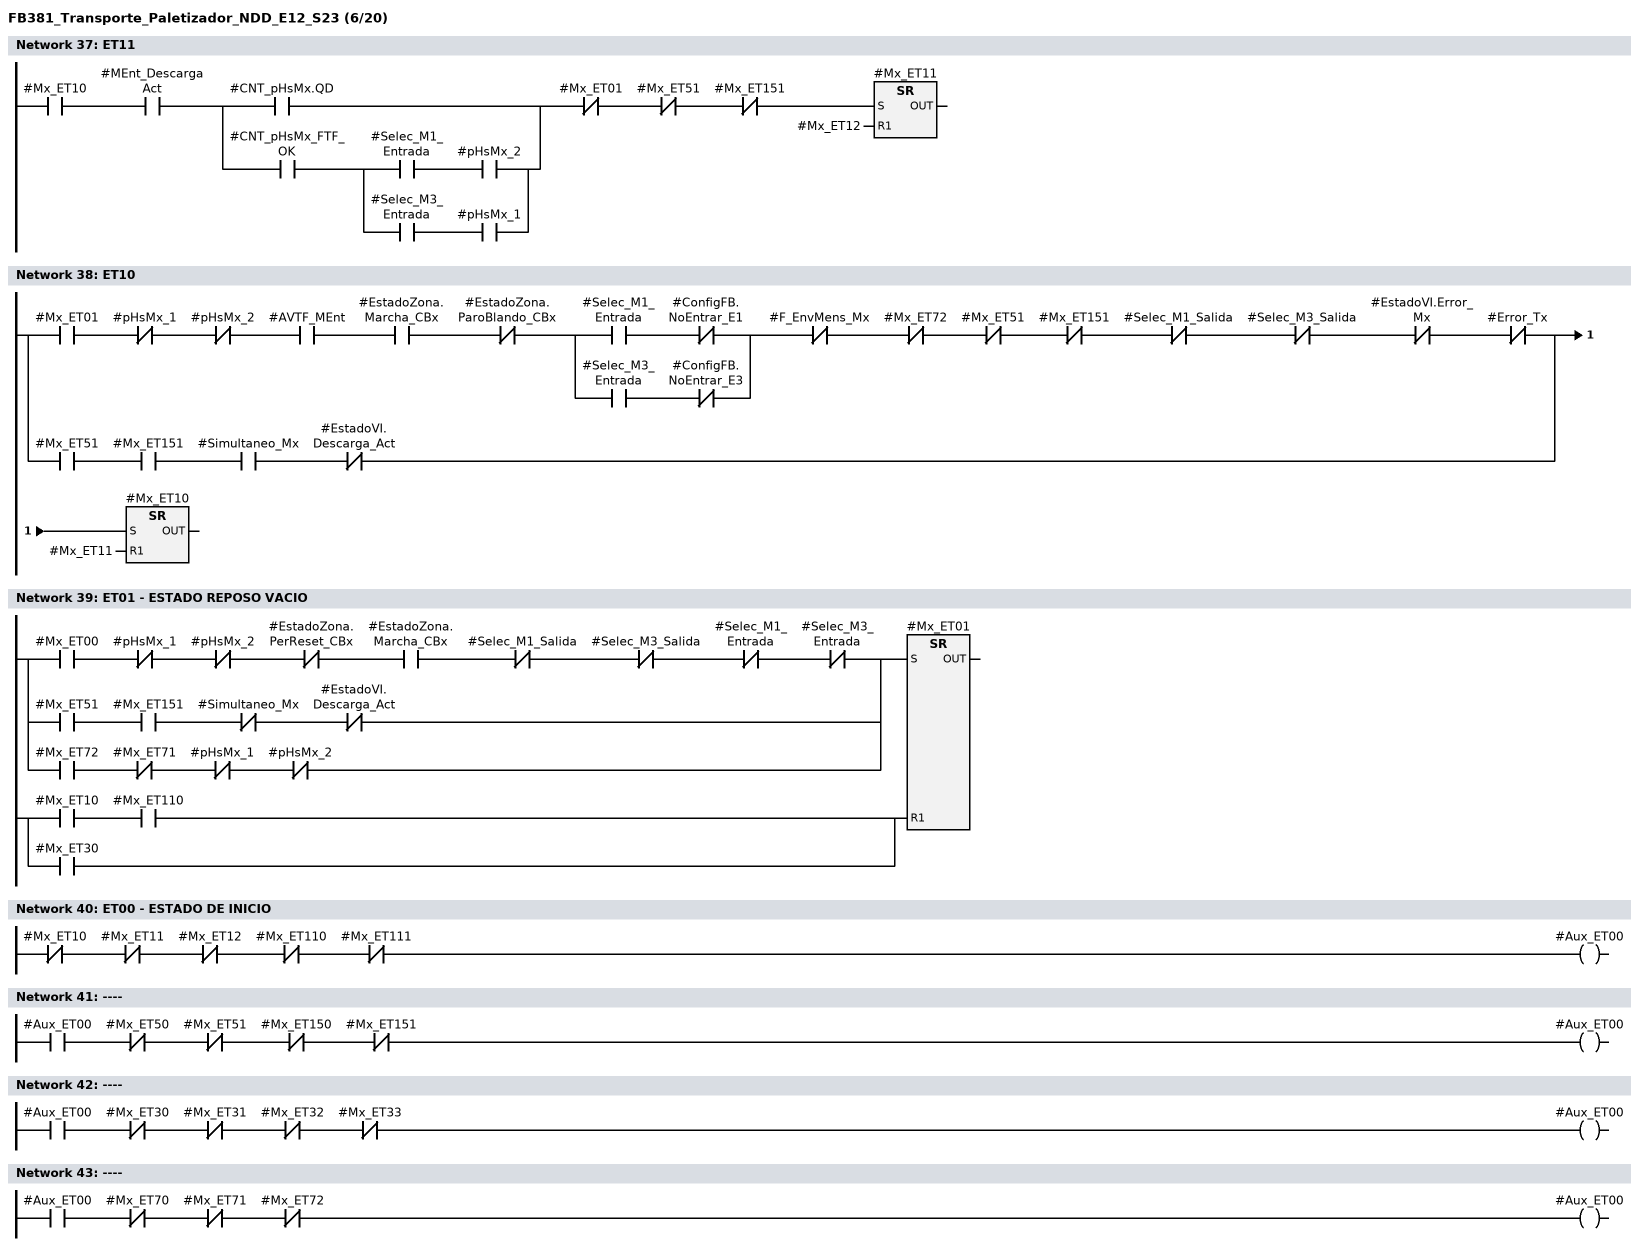
   RUNG wire#powerrail
      Contact( #Mx_ET10 )
      Contact( #MEnt_DescargaAct )
      wire#w1
      Contact( #CNT_pHsMx.QD )
      wire#w2
      I_Contact( #Mx_ET01 )
      I_Contact( #Mx_ET51 )
      I_Contact( #Mx_ET151 )
      S_SR(operand := #Mx_ET11, r1 := #Mx_ET12)
   END_RUNG
   RUNG wire#w1
      Contact( #CNT_pHsMx_FTF_OK )
      wire#w3
      Contact( #Selec_M1_Entrada )
      Contact( #pHsMx_2 )
   END_RUNG wire#w2
   RUNG wire#w3
      Contact( #Selec_M3_Entrada )
      Contact( #pHsMx_1 )
   END_RUNG wire#w2
   // the same network as SCL:
   IF #Mx_ET10 AND #MEnt_DescargaAct AND (#CNT_pHsMx.QD OR (#CNT_pHsMx_FTF_OK AND ((#Selec_M1_Entrada AND #pHsMx_2) OR (#Selec_M3_Entrada AND #pHsMx_1)))) AND NOT #Mx_ET01 AND NOT #Mx_ET51 AND NOT #Mx_ET151 THEN
       #Mx_ET11 := TRUE;   // SR flip-flop
   END_IF;
   IF #Mx_ET12 THEN #Mx_ET11 := FALSE; END_IF;
END_REGION

REGION Network 38: ET10
   RUNG wire#powerrail
      Contact( #Mx_ET01 )
      I_Contact( #pHsMx_1 )
      I_Contact( #pHsMx_2 )
      Contact( #AVTF_MEnt )
      Contact( #EstadoZona.Marcha_CBx )
      I_Contact( #EstadoZona.ParoBlando_CBx )
      wire#w1
      Contact( #Selec_M1_Entrada )
      I_Contact( #ConfigFB.NoEntrar_E1 )
      wire#w2
      I_Contact( #F_EnvMens_Mx )
      I_Contact( #Mx_ET72 )
      I_Contact( #Mx_ET51 )
      I_Contact( #Mx_ET151 )
      I_Contact( #Selec_M1_Salida )
      I_Contact( #Selec_M3_Salida )
      I_Contact( #EstadoVI.Error_Mx )
      I_Contact( #Error_Tx )
      wire#w3
      S_SR(operand := #Mx_ET10, r1 := #Mx_ET11)
   END_RUNG
   RUNG wire#w1
      Contact( #Selec_M3_Entrada )
      I_Contact( #ConfigFB.NoEntrar_E3 )
   END_RUNG wire#w2
   RUNG wire#powerrail
      Contact( #Mx_ET51 )
      Contact( #Mx_ET151 )
      Contact( #Simultaneo_Mx )
      I_Contact( #EstadoVI.Descarga_Act )
   END_RUNG wire#w3
   // the same network as SCL:
   IF (#Mx_ET01 AND NOT #pHsMx_1 AND NOT #pHsMx_2 AND #AVTF_MEnt AND #EstadoZona.Marcha_CBx AND NOT #EstadoZona.ParoBlando_CBx AND ((#Selec_M1_Entrada AND NOT #ConfigFB.NoEntrar_E1) OR (#Selec_M3_Entrada AND NOT #ConfigFB.NoEntrar_E3)) AND NOT #F_EnvMens_Mx AND NOT #Mx_ET72 AND NOT #Mx_ET51 AND NOT #Mx_ET151 AND NOT #Selec_M1_Salida AND NOT #Selec_M3_Salida AND NOT #EstadoVI.Error_Mx AND NOT #Error_Tx) OR (#Mx_ET51 AND #Mx_ET151 AND #Simultaneo_Mx AND NOT #EstadoVI.Descarga_Act) THEN
       #Mx_ET10 := TRUE;   // SR flip-flop
   END_IF;
   IF #Mx_ET11 THEN #Mx_ET10 := FALSE; END_IF;
END_REGION

REGION Network 39: ET01 - ESTADO REPOSO VACIO
   RUNG wire#powerrail
      Contact( #Mx_ET00 )
      I_Contact( #pHsMx_1 )
      I_Contact( #pHsMx_2 )
      I_Contact( #EstadoZona.PerReset_CBx )
      Contact( #EstadoZona.Marcha_CBx )
      I_Contact( #Selec_M1_Salida )
      I_Contact( #Selec_M3_Salida )
      I_Contact( #Selec_M1_Entrada )
      I_Contact( #Selec_M3_Entrada )
      wire#w1
      S_SR(operand := #Mx_ET01, r1 := wire#w2)
   END_RUNG
   RUNG wire#powerrail
      Contact( #Mx_ET51 )
      Contact( #Mx_ET151 )
      I_Contact( #Simultaneo_Mx )
      I_Contact( #EstadoVI.Descarga_Act )
   END_RUNG wire#w1
   RUNG wire#powerrail
      Contact( #Mx_ET72 )
      I_Contact( #Mx_ET71 )
      I_Contact( #pHsMx_1 )
      I_Contact( #pHsMx_2 )
   END_RUNG wire#w1
   RUNG wire#powerrail
      Contact( #Mx_ET10 )
      Contact( #Mx_ET110 )
   END_RUNG wire#w2
   RUNG wire#powerrail
      Contact( #Mx_ET30 )
   END_RUNG wire#w2
   // the same network as SCL:
   IF (#Mx_ET00 AND NOT #pHsMx_1 AND NOT #pHsMx_2 AND NOT #EstadoZona.PerReset_CBx AND #EstadoZona.Marcha_CBx AND NOT #Selec_M1_Salida AND NOT #Selec_M3_Salida AND NOT #Selec_M1_Entrada AND NOT #Selec_M3_Entrada) OR (#Mx_ET51 AND #Mx_ET151 AND NOT #Simultaneo_Mx AND NOT #EstadoVI.Descarga_Act) OR (#Mx_ET72 AND NOT #Mx_ET71 AND NOT #pHsMx_1 AND NOT #pHsMx_2) THEN
       #Mx_ET01 := TRUE;   // SR flip-flop
   END_IF;
   IF (#Mx_ET10 AND #Mx_ET110) OR #Mx_ET30 THEN #Mx_ET01 := FALSE; END_IF;
END_REGION

REGION Network 40: ET00 - ESTADO DE INICIO
   RUNG wire#powerrail
      I_Contact( #Mx_ET10 )
      I_Contact( #Mx_ET11 )
      I_Contact( #Mx_ET12 )
      I_Contact( #Mx_ET110 )
      I_Contact( #Mx_ET111 )
      Coil( #Aux_ET00 )
   END_RUNG
   // the same network as SCL:
   #Aux_ET00 := NOT #Mx_ET10 AND NOT #Mx_ET11 AND NOT #Mx_ET12 AND NOT #Mx_ET110 AND NOT #Mx_ET111;
END_REGION

REGION Network 41: ----
   RUNG wire#powerrail
      Contact( #Aux_ET00 )
      I_Contact( #Mx_ET50 )
      I_Contact( #Mx_ET51 )
      I_Contact( #Mx_ET150 )
      I_Contact( #Mx_ET151 )
      Coil( #Aux_ET00 )
   END_RUNG
   // the same network as SCL:
   #Aux_ET00 := #Aux_ET00 AND NOT #Mx_ET50 AND NOT #Mx_ET51 AND NOT #Mx_ET150 AND NOT #Mx_ET151;
END_REGION

REGION Network 42: ----
   RUNG wire#powerrail
      Contact( #Aux_ET00 )
      I_Contact( #Mx_ET30 )
      I_Contact( #Mx_ET31 )
      I_Contact( #Mx_ET32 )
      I_Contact( #Mx_ET33 )
      Coil( #Aux_ET00 )
   END_RUNG
   // the same network as SCL:
   #Aux_ET00 := #Aux_ET00 AND NOT #Mx_ET30 AND NOT #Mx_ET31 AND NOT #Mx_ET32 AND NOT #Mx_ET33;
END_REGION

REGION Network 43: ----
   RUNG wire#powerrail
      Contact( #Aux_ET00 )
      I_Contact( #Mx_ET70 )
      I_Contact( #Mx_ET71 )
      I_Contact( #Mx_ET72 )
      Coil( #Aux_ET00 )
   END_RUNG
   // the same network as SCL:
   #Aux_ET00 := #Aux_ET00 AND NOT #Mx_ET70 AND NOT #Mx_ET71 AND NOT #Mx_ET72;
END_REGION

REGION Network 44: ----
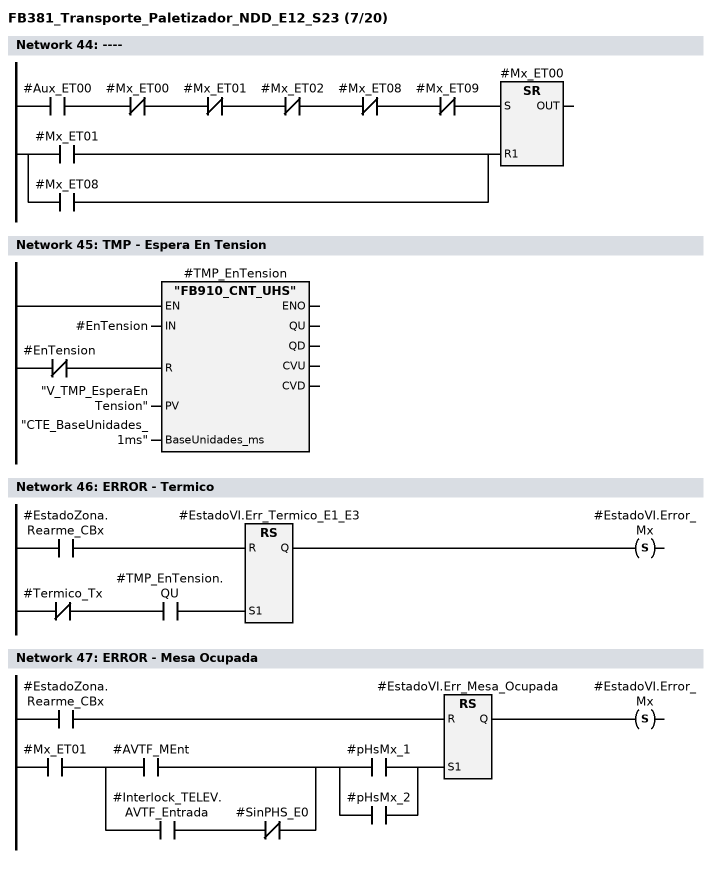
   RUNG wire#powerrail
      Contact( #Aux_ET00 )
      I_Contact( #Mx_ET00 )
      I_Contact( #Mx_ET01 )
      I_Contact( #Mx_ET02 )
      I_Contact( #Mx_ET08 )
      I_Contact( #Mx_ET09 )
      S_SR(operand := #Mx_ET00, r1 := wire#w1)
   END_RUNG
   RUNG wire#powerrail
      Contact( #Mx_ET01 )
   END_RUNG wire#w1
   RUNG wire#powerrail
      Contact( #Mx_ET08 )
   END_RUNG wire#w1
   // the same network as SCL:
   IF #Aux_ET00 AND NOT #Mx_ET00 AND NOT #Mx_ET01 AND NOT #Mx_ET02 AND NOT #Mx_ET08 AND NOT #Mx_ET09 THEN
       #Mx_ET00 := TRUE;   // SR flip-flop
   END_IF;
   IF #Mx_ET01 OR #Mx_ET08 THEN #Mx_ET00 := FALSE; END_IF;
END_REGION

REGION Network 45: TMP - Espera En Tension
   RUNG wire#powerrail
      #TMP_EnTension(R := wire#w1, IN := #EnTension, PV := "V_TMP_EsperaEnTension", BaseUnidades_ms := "CTE_BaseUnidades_1ms", QU =>, QD =>, CVU =>, CVD =>)
   END_RUNG
   RUNG wire#powerrail
      I_Contact( #EnTension )
   END_RUNG wire#w1
   // the same network as SCL:
   #TMP_EnTension(IN := #EnTension,   // "FB910_CNT_UHS"
                  R := NOT #EnTension,
                  PV := "V_TMP_EsperaEnTension",
                  BaseUnidades_ms := "CTE_BaseUnidades_1ms");
END_REGION

REGION Network 46: ERROR - Termico
   RUNG wire#powerrail
      Contact( #EstadoZona.Rearme_CBx )
      S_RS(operand := #EstadoVI.Err_Termico_E1_E3, s1 := wire#w1)
      S_Coil( #EstadoVI.Error_Mx )
   END_RUNG
   RUNG wire#powerrail
      I_Contact( #Termico_Tx )
      Contact( #TMP_EnTension.QU )
   END_RUNG wire#w1
   // the same network as SCL:
   IF #EstadoZona.Rearme_CBx THEN
       #EstadoVI.Err_Termico_E1_E3 := FALSE;   // RS flip-flop
   END_IF;
   IF NOT #Termico_Tx AND #TMP_EnTension.QU THEN #EstadoVI.Err_Termico_E1_E3 := TRUE; END_IF;
   IF #EstadoVI.Err_Termico_E1_E3 THEN #EstadoVI.Error_Mx := TRUE; END_IF;
END_REGION

REGION Network 47: ERROR - Mesa Ocupada
   RUNG wire#powerrail
      Contact( #EstadoZona.Rearme_CBx )
      S_RS(operand := #EstadoVI.Err_Mesa_Ocupada, s1 := wire#w3)
      S_Coil( #EstadoVI.Error_Mx )
   END_RUNG
   RUNG wire#powerrail
      Contact( #Mx_ET01 )
      wire#w1
      Contact( #AVTF_MEnt )
      wire#w2
      Contact( #pHsMx_1 )
   END_RUNG wire#w3
   RUNG wire#w1
      Contact( #Interlock_TELEV.AVTF_Entrada )
      I_Contact( #SinPHS_E0 )
   END_RUNG wire#w2
   RUNG wire#w2
      Contact( #pHsMx_2 )
   END_RUNG wire#w3
   // the same network as SCL:
   IF #EstadoZona.Rearme_CBx THEN
       #EstadoVI.Err_Mesa_Ocupada := FALSE;   // RS flip-flop
   END_IF;
   IF #Mx_ET01 AND (#AVTF_MEnt OR (#Interlock_TELEV.AVTF_Entrada AND NOT #SinPHS_E0)) AND (#pHsMx_1 OR #pHsMx_2) THEN
       #EstadoVI.Err_Mesa_Ocupada := TRUE;
   END_IF;
   IF #EstadoVI.Err_Mesa_Ocupada THEN #EstadoVI.Error_Mx := TRUE; END_IF;
END_REGION

REGION Network 48: CNT - ERROR - Arrastre
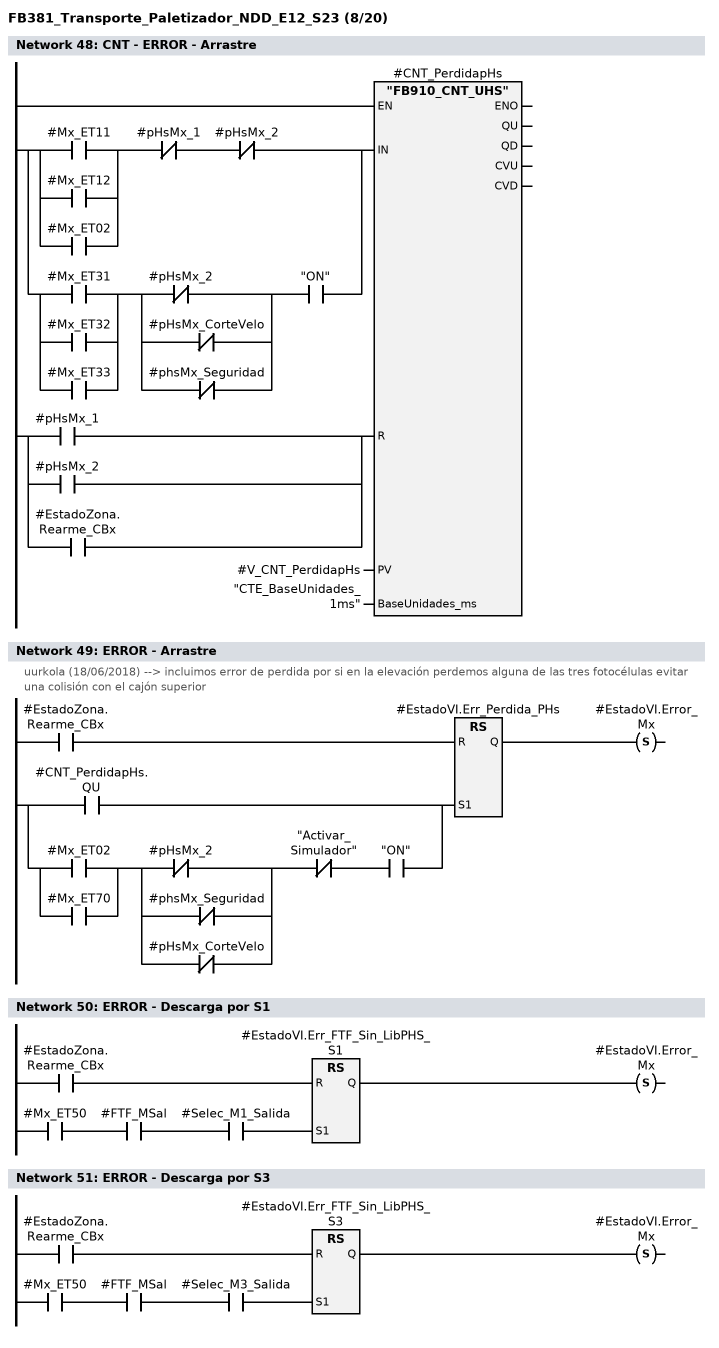
   RUNG wire#powerrail
      #CNT_PerdidapHs(IN := wire#w4, R := wire#w5, PV := #V_CNT_PerdidapHs, BaseUnidades_ms := "CTE_BaseUnidades_1ms", QU =>, QD =>, CVU =>, CVD =>)
   END_RUNG
   RUNG wire#powerrail
      Contact( #Mx_ET11 )
      wire#w1
      I_Contact( #pHsMx_1 )
      I_Contact( #pHsMx_2 )
   END_RUNG wire#w4
   RUNG wire#powerrail
      Contact( #Mx_ET12 )
   END_RUNG wire#w1
   RUNG wire#powerrail
      Contact( #Mx_ET02 )
   END_RUNG wire#w1
   RUNG wire#powerrail
      Contact( #Mx_ET31 )
      wire#w2
      I_Contact( #pHsMx_2 )
      wire#w3
      Contact( "ON" )
   END_RUNG wire#w4
   RUNG wire#powerrail
      Contact( #Mx_ET32 )
   END_RUNG wire#w2
   RUNG wire#powerrail
      Contact( #Mx_ET33 )
   END_RUNG wire#w2
   RUNG wire#w2
      I_Contact( #pHsMx_CorteVelo )
   END_RUNG wire#w3
   RUNG wire#w2
      I_Contact( #phsMx_Seguridad )
   END_RUNG wire#w3
   RUNG wire#powerrail
      Contact( #pHsMx_1 )
   END_RUNG wire#w5
   RUNG wire#powerrail
      Contact( #pHsMx_2 )
   END_RUNG wire#w5
   RUNG wire#powerrail
      Contact( #EstadoZona.Rearme_CBx )
   END_RUNG wire#w5
   // the same network as SCL:
   #CNT_PerdidapHs(IN := ((#Mx_ET11 OR #Mx_ET12 OR #Mx_ET02) AND NOT #pHsMx_1 AND NOT #pHsMx_2) OR ((#Mx_ET31 OR #Mx_ET32 OR #Mx_ET33) AND (NOT #pHsMx_2 OR NOT #pHsMx_CorteVelo OR NOT #phsMx_Seguridad) AND "ON"),   // "FB910_CNT_UHS"
                   R := #pHsMx_1 OR #pHsMx_2 OR #EstadoZona.Rearme_CBx,
                   PV := #V_CNT_PerdidapHs,
                   BaseUnidades_ms := "CTE_BaseUnidades_1ms");
END_REGION

REGION Network 49: ERROR - Arrastre
   // uurkola (18/06/2018) --> incluimos error de perdida por si en la elevación perdemos alguna de las tres fotocélulas evitar una colisión con el cajón superior
   RUNG wire#powerrail
      Contact( #EstadoZona.Rearme_CBx )
      S_RS(operand := #EstadoVI.Err_Perdida_PHs, s1 := wire#w3)
      S_Coil( #EstadoVI.Error_Mx )
   END_RUNG
   RUNG wire#powerrail
      Contact( #CNT_PerdidapHs.QU )
   END_RUNG wire#w3
   RUNG wire#powerrail
      Contact( #Mx_ET02 )
      wire#w1
      I_Contact( #pHsMx_2 )
      wire#w2
      I_Contact( "Activar_Simulador" )
      Contact( "ON" )
   END_RUNG wire#w3
   RUNG wire#powerrail
      Contact( #Mx_ET70 )
   END_RUNG wire#w1
   RUNG wire#w1
      I_Contact( #phsMx_Seguridad )
   END_RUNG wire#w2
   RUNG wire#w1
      I_Contact( #pHsMx_CorteVelo )
   END_RUNG wire#w2
   // the same network as SCL:
   IF #EstadoZona.Rearme_CBx THEN
       #EstadoVI.Err_Perdida_PHs := FALSE;   // RS flip-flop
   END_IF;
   IF #CNT_PerdidapHs.QU OR ((#Mx_ET02 OR #Mx_ET70) AND (NOT #pHsMx_2 OR NOT #phsMx_Seguridad OR NOT #pHsMx_CorteVelo) AND NOT "Activar_Simulador" AND "ON") THEN
       #EstadoVI.Err_Perdida_PHs := TRUE;
   END_IF;
   IF #EstadoVI.Err_Perdida_PHs THEN #EstadoVI.Error_Mx := TRUE; END_IF;
END_REGION

REGION Network 50: ERROR - Descarga por S1
   RUNG wire#powerrail
      Contact( #EstadoZona.Rearme_CBx )
      S_RS(operand := #EstadoVI.Err_FTF_Sin_LibPHS_S1, s1 := wire#w1)
      S_Coil( #EstadoVI.Error_Mx )
   END_RUNG
   RUNG wire#powerrail
      Contact( #Mx_ET50 )
      Contact( #FTF_MSal )
      Contact( #Selec_M1_Salida )
   END_RUNG wire#w1
   // the same network as SCL:
   IF #EstadoZona.Rearme_CBx THEN
       #EstadoVI.Err_FTF_Sin_LibPHS_S1 := FALSE;   // RS flip-flop
   END_IF;
   IF #Mx_ET50 AND #FTF_MSal AND #Selec_M1_Salida THEN #EstadoVI.Err_FTF_Sin_LibPHS_S1 := TRUE; END_IF;
   IF #EstadoVI.Err_FTF_Sin_LibPHS_S1 THEN #EstadoVI.Error_Mx := TRUE; END_IF;
END_REGION

REGION Network 51: ERROR - Descarga por S3
   RUNG wire#powerrail
      Contact( #EstadoZona.Rearme_CBx )
      S_RS(operand := #EstadoVI.Err_FTF_Sin_LibPHS_S3, s1 := wire#w1)
      S_Coil( #EstadoVI.Error_Mx )
   END_RUNG
   RUNG wire#powerrail
      Contact( #Mx_ET50 )
      Contact( #FTF_MSal )
      Contact( #Selec_M3_Salida )
   END_RUNG wire#w1
   // the same network as SCL:
   IF #EstadoZona.Rearme_CBx THEN
       #EstadoVI.Err_FTF_Sin_LibPHS_S3 := FALSE;   // RS flip-flop
   END_IF;
   IF #Mx_ET50 AND #FTF_MSal AND #Selec_M3_Salida THEN #EstadoVI.Err_FTF_Sin_LibPHS_S3 := TRUE; END_IF;
   IF #EstadoVI.Err_FTF_Sin_LibPHS_S3 THEN #EstadoVI.Error_Mx := TRUE; END_IF;
END_REGION

REGION Network 52: TMP - ERROR - TimeOut Avance
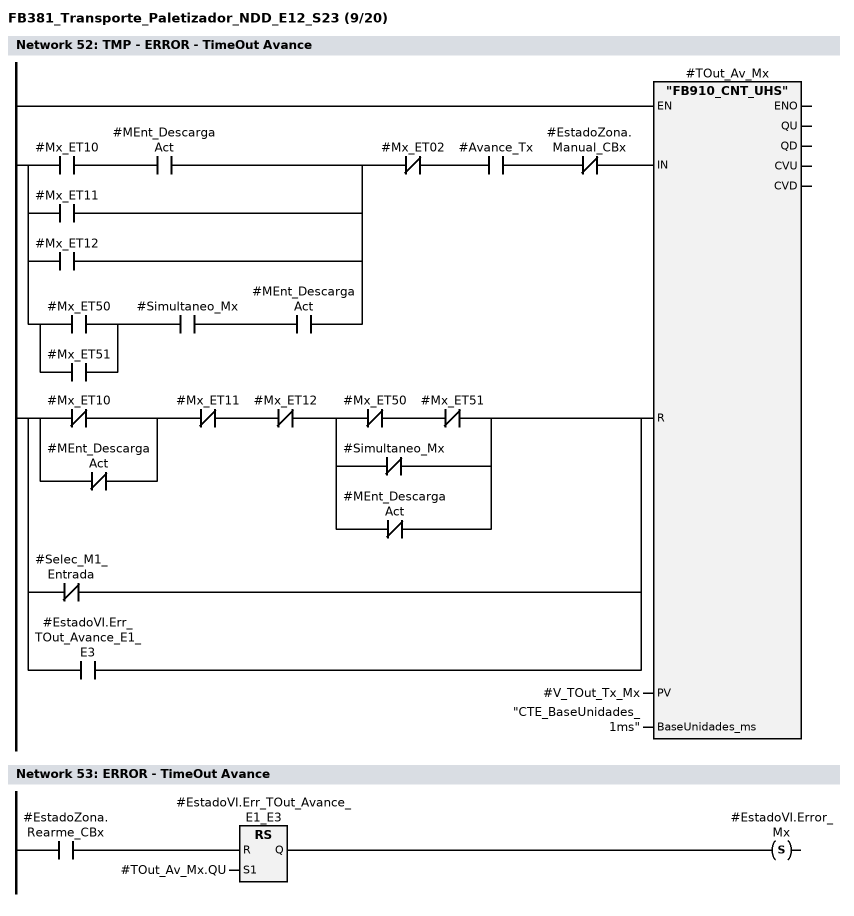
   RUNG wire#powerrail
      #TOut_Av_Mx(IN := wire#w3, R := wire#w6, PV := #V_TOut_Tx_Mx, BaseUnidades_ms := "CTE_BaseUnidades_1ms", QU =>, QD =>, CVU =>, CVD =>)
   END_RUNG
   RUNG wire#powerrail
      Contact( #Mx_ET10 )
      Contact( #MEnt_DescargaAct )
      wire#w1
      I_Contact( #Mx_ET02 )
      Contact( #Avance_Tx )
      I_Contact( #EstadoZona.Manual_CBx )
   END_RUNG wire#w3
   RUNG wire#powerrail
      Contact( #Mx_ET11 )
   END_RUNG wire#w1
   RUNG wire#powerrail
      Contact( #Mx_ET12 )
   END_RUNG wire#w1
   RUNG wire#powerrail
      Contact( #Mx_ET50 )
      wire#w2
      Contact( #Simultaneo_Mx )
      Contact( #MEnt_DescargaAct )
   END_RUNG wire#w1
   RUNG wire#powerrail
      Contact( #Mx_ET51 )
   END_RUNG wire#w2
   RUNG wire#powerrail
      I_Contact( #Mx_ET10 )
      wire#w4
      I_Contact( #Mx_ET11 )
      I_Contact( #Mx_ET12 )
      wire#w5
      I_Contact( #Mx_ET50 )
      I_Contact( #Mx_ET51 )
   END_RUNG wire#w6
   RUNG wire#powerrail
      I_Contact( #MEnt_DescargaAct )
   END_RUNG wire#w4
   RUNG wire#w5
      I_Contact( #Simultaneo_Mx )
   END_RUNG wire#w6
   RUNG wire#w5
      I_Contact( #MEnt_DescargaAct )
   END_RUNG wire#w6
   RUNG wire#powerrail
      I_Contact( #Selec_M1_Entrada )
   END_RUNG wire#w6
   RUNG wire#powerrail
      Contact( #EstadoVI.Err_TOut_Avance_E1_E3 )
   END_RUNG wire#w6
   // the same network as SCL:
   #TOut_Av_Mx(IN := ((#Mx_ET10 AND #MEnt_DescargaAct) OR #Mx_ET11 OR #Mx_ET12 OR ((#Mx_ET50 OR #Mx_ET51) AND #Simultaneo_Mx AND #MEnt_DescargaAct)) AND NOT #Mx_ET02 AND #Avance_Tx AND NOT #EstadoZona.Manual_CBx,   // "FB910_CNT_UHS"
               R := ((NOT #Mx_ET10 OR NOT #MEnt_DescargaAct) AND NOT #Mx_ET11 AND NOT #Mx_ET12 AND ((NOT #Mx_ET50 AND NOT #Mx_ET51) OR NOT #Simultaneo_Mx OR NOT #MEnt_DescargaAct)) OR NOT #Selec_M1_Entrada OR #EstadoVI.Err_TOut_Avance_E1_E3,
               PV := #V_TOut_Tx_Mx,
               BaseUnidades_ms := "CTE_BaseUnidades_1ms");
END_REGION

REGION Network 53: ERROR - TimeOut Avance
   RUNG wire#powerrail
      Contact( #EstadoZona.Rearme_CBx )
      S_RS(operand := #EstadoVI.Err_TOut_Avance_E1_E3, s1 := #TOut_Av_Mx.QU)
      S_Coil( #EstadoVI.Error_Mx )
   END_RUNG
   // the same network as SCL:
   IF #EstadoZona.Rearme_CBx THEN
       #EstadoVI.Err_TOut_Avance_E1_E3 := FALSE;   // RS flip-flop
   END_IF;
   IF #TOut_Av_Mx.QU THEN #EstadoVI.Err_TOut_Avance_E1_E3 := TRUE; END_IF;
   IF #EstadoVI.Err_TOut_Avance_E1_E3 THEN #EstadoVI.Error_Mx := TRUE; END_IF;
END_REGION

REGION Network 54: TMP - ERROR - TimeOut Retroceso
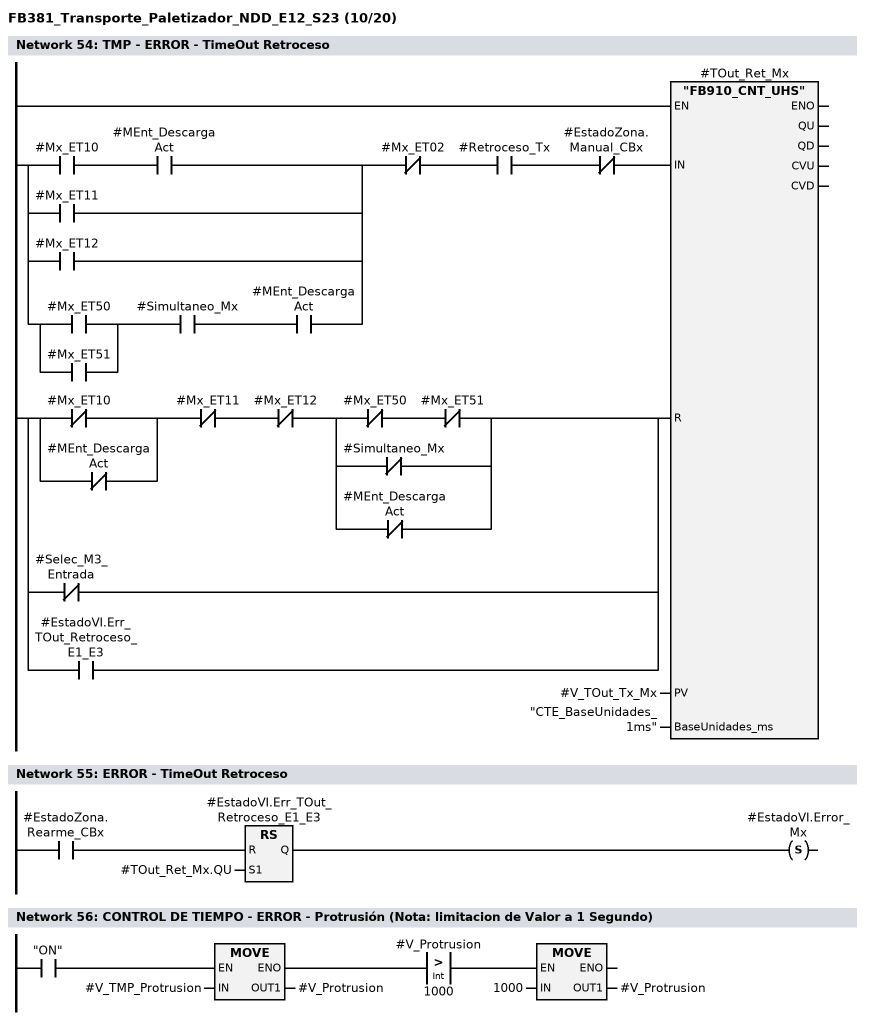
   RUNG wire#powerrail
      #TOut_Ret_Mx(IN := wire#w3, R := wire#w6, PV := #V_TOut_Tx_Mx, BaseUnidades_ms := "CTE_BaseUnidades_1ms", QU =>, QD =>, CVU =>, CVD =>)
   END_RUNG
   RUNG wire#powerrail
      Contact( #Mx_ET10 )
      Contact( #MEnt_DescargaAct )
      wire#w1
      I_Contact( #Mx_ET02 )
      Contact( #Retroceso_Tx )
      I_Contact( #EstadoZona.Manual_CBx )
   END_RUNG wire#w3
   RUNG wire#powerrail
      Contact( #Mx_ET11 )
   END_RUNG wire#w1
   RUNG wire#powerrail
      Contact( #Mx_ET12 )
   END_RUNG wire#w1
   RUNG wire#powerrail
      Contact( #Mx_ET50 )
      wire#w2
      Contact( #Simultaneo_Mx )
      Contact( #MEnt_DescargaAct )
   END_RUNG wire#w1
   RUNG wire#powerrail
      Contact( #Mx_ET51 )
   END_RUNG wire#w2
   RUNG wire#powerrail
      I_Contact( #Mx_ET10 )
      wire#w4
      I_Contact( #Mx_ET11 )
      I_Contact( #Mx_ET12 )
      wire#w5
      I_Contact( #Mx_ET50 )
      I_Contact( #Mx_ET51 )
   END_RUNG wire#w6
   RUNG wire#powerrail
      I_Contact( #MEnt_DescargaAct )
   END_RUNG wire#w4
   RUNG wire#w5
      I_Contact( #Simultaneo_Mx )
   END_RUNG wire#w6
   RUNG wire#w5
      I_Contact( #MEnt_DescargaAct )
   END_RUNG wire#w6
   RUNG wire#powerrail
      I_Contact( #Selec_M3_Entrada )
   END_RUNG wire#w6
   RUNG wire#powerrail
      Contact( #EstadoVI.Err_TOut_Retroceso_E1_E3 )
   END_RUNG wire#w6
   // the same network as SCL:
   #TOut_Ret_Mx(IN := ((#Mx_ET10 AND #MEnt_DescargaAct) OR #Mx_ET11 OR #Mx_ET12 OR ((#Mx_ET50 OR #Mx_ET51) AND #Simultaneo_Mx AND #MEnt_DescargaAct)) AND NOT #Mx_ET02 AND #Retroceso_Tx AND NOT #EstadoZona.Manual_CBx,   // "FB910_CNT_UHS"
                R := ((NOT #Mx_ET10 OR NOT #MEnt_DescargaAct) AND NOT #Mx_ET11 AND NOT #Mx_ET12 AND ((NOT #Mx_ET50 AND NOT #Mx_ET51) OR NOT #Simultaneo_Mx OR NOT #MEnt_DescargaAct)) OR NOT #Selec_M3_Entrada OR #EstadoVI.Err_TOut_Retroceso_E1_E3,
                PV := #V_TOut_Tx_Mx,
                BaseUnidades_ms := "CTE_BaseUnidades_1ms");
END_REGION

REGION Network 55: ERROR - TimeOut Retroceso
   RUNG wire#powerrail
      Contact( #EstadoZona.Rearme_CBx )
      S_RS(operand := #EstadoVI.Err_TOut_Retroceso_E1_E3, s1 := #TOut_Ret_Mx.QU)
      S_Coil( #EstadoVI.Error_Mx )
   END_RUNG
   // the same network as SCL:
   IF #EstadoZona.Rearme_CBx THEN
       #EstadoVI.Err_TOut_Retroceso_E1_E3 := FALSE;   // RS flip-flop
   END_IF;
   IF #TOut_Ret_Mx.QU THEN #EstadoVI.Err_TOut_Retroceso_E1_E3 := TRUE; END_IF;
   IF #EstadoVI.Err_TOut_Retroceso_E1_E3 THEN #EstadoVI.Error_Mx := TRUE; END_IF;
END_REGION

REGION Network 56: CONTROL DE TIEMPO - ERROR - Protrusión (Nota: limitacion de Valor a 1 Segundo)
   RUNG wire#powerrail
      Contact( "ON" )
      Move(in := #V_TMP_Protrusion, out1 => #V_Protrusion)
      { S7_Templates := "SrcType := Int" } GT_Contact(in1 := #V_Protrusion, in2 := 1000)
      Move(in := 1000, out1 => #V_Protrusion)
   END_RUNG
   // the same network as SCL:
   IF "ON" THEN #V_Protrusion := #V_TMP_Protrusion; END_IF;
   IF "ON" AND (#V_Protrusion > 1000) THEN #V_Protrusion := 1000; END_IF;
END_REGION

REGION Network 57: TMP - ERROR - Protrusión
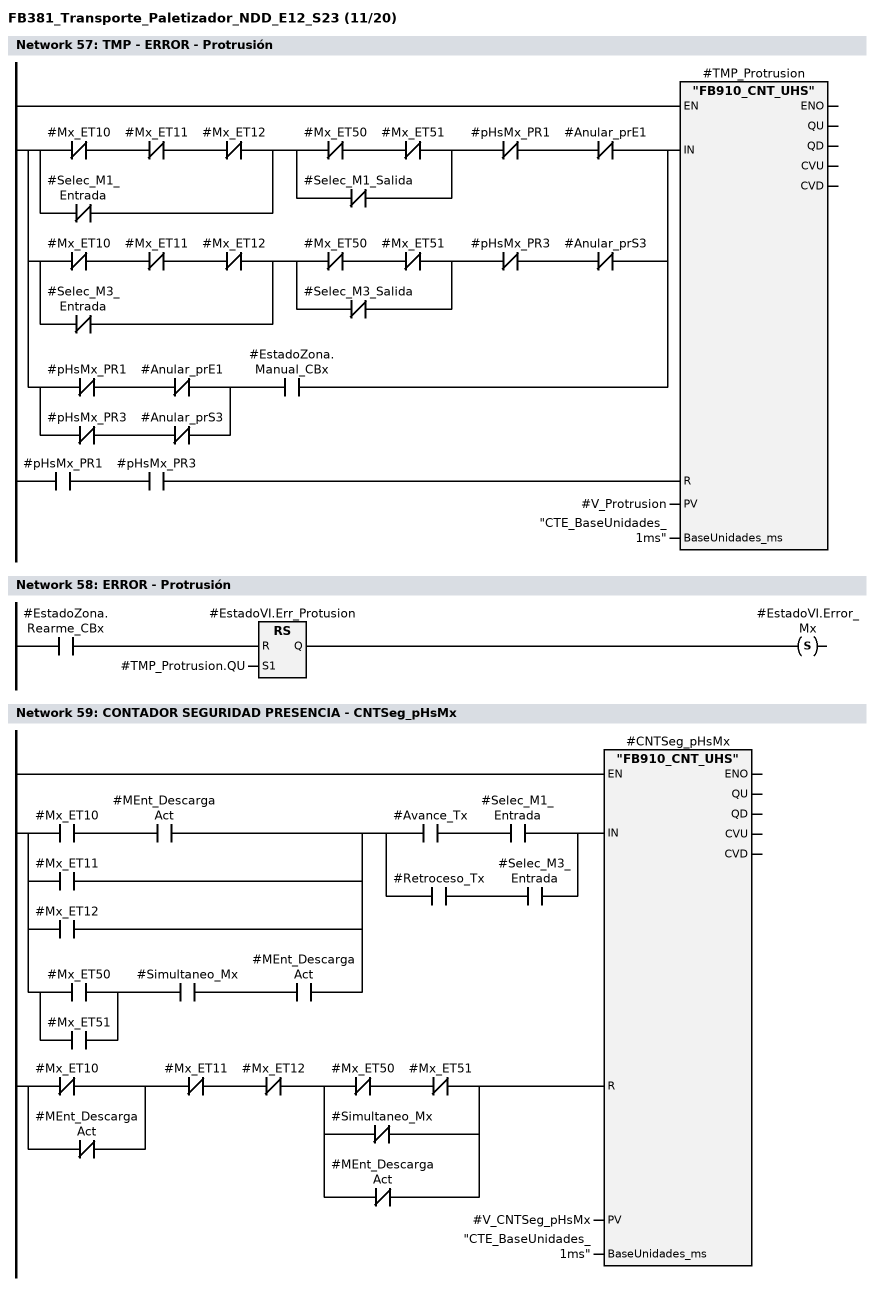
   RUNG wire#powerrail
      #TMP_Protrusion(IN := wire#w6, R := wire#w7, PV := #V_Protrusion, BaseUnidades_ms := "CTE_BaseUnidades_1ms", QU =>, QD =>, CVU =>, CVD =>)
   END_RUNG
   RUNG wire#powerrail
      I_Contact( #Mx_ET10 )
      I_Contact( #Mx_ET11 )
      I_Contact( #Mx_ET12 )
      wire#w1
      I_Contact( #Mx_ET50 )
      I_Contact( #Mx_ET51 )
      wire#w2
      I_Contact( #pHsMx_PR1 )
      I_Contact( #Anular_prE1 )
   END_RUNG wire#w6
   RUNG wire#powerrail
      I_Contact( #Selec_M1_Entrada )
   END_RUNG wire#w1
   RUNG wire#w1
      I_Contact( #Selec_M1_Salida )
   END_RUNG wire#w2
   RUNG wire#powerrail
      I_Contact( #Mx_ET10 )
      I_Contact( #Mx_ET11 )
      I_Contact( #Mx_ET12 )
      wire#w3
      I_Contact( #Mx_ET50 )
      I_Contact( #Mx_ET51 )
      wire#w4
      I_Contact( #pHsMx_PR3 )
      I_Contact( #Anular_prS3 )
   END_RUNG wire#w6
   RUNG wire#powerrail
      I_Contact( #Selec_M3_Entrada )
   END_RUNG wire#w3
   RUNG wire#w3
      I_Contact( #Selec_M3_Salida )
   END_RUNG wire#w4
   RUNG wire#powerrail
      I_Contact( #pHsMx_PR1 )
      I_Contact( #Anular_prE1 )
      wire#w5
      Contact( #EstadoZona.Manual_CBx )
   END_RUNG wire#w6
   RUNG wire#powerrail
      I_Contact( #pHsMx_PR3 )
      I_Contact( #Anular_prS3 )
   END_RUNG wire#w5
   RUNG wire#powerrail
      Contact( #pHsMx_PR1 )
      Contact( #pHsMx_PR3 )
   END_RUNG wire#w7
   // the same network as SCL:
   #TMP_Protrusion(IN := (((NOT #Mx_ET10 AND NOT #Mx_ET11 AND NOT #Mx_ET12) OR NOT #Selec_M1_Entrada) AND ((NOT #Mx_ET50 AND NOT #Mx_ET51) OR NOT #Selec_M1_Salida) AND NOT #pHsMx_PR1 AND NOT #Anular_prE1) OR (((NOT #Mx_ET10 AND NOT #Mx_ET11 AND NOT #Mx_ET12) OR NOT #Selec_M3_Entrada) AND ((NOT #Mx_ET50 AND NOT #Mx_ET51) OR NOT #Selec_M3_Salida) AND NOT #pHsMx_PR3 AND NOT #Anular_prS3) OR (((NOT #pHsMx_PR1 AND NOT #Anular_prE1) OR (NOT #pHsMx_PR3 AND NOT #Anular_prS3)) AND #EstadoZona.Manual_CBx),   // "FB910_CNT_UHS"
                   R := #pHsMx_PR1 AND #pHsMx_PR3,
                   PV := #V_Protrusion,
                   BaseUnidades_ms := "CTE_BaseUnidades_1ms");
END_REGION

REGION Network 58: ERROR - Protrusión
   RUNG wire#powerrail
      Contact( #EstadoZona.Rearme_CBx )
      S_RS(operand := #EstadoVI.Err_Protusion, s1 := #TMP_Protrusion.QU)
      S_Coil( #EstadoVI.Error_Mx )
   END_RUNG
   // the same network as SCL:
   IF #EstadoZona.Rearme_CBx THEN
       #EstadoVI.Err_Protusion := FALSE;   // RS flip-flop
   END_IF;
   IF #TMP_Protrusion.QU THEN #EstadoVI.Err_Protusion := TRUE; END_IF;
   IF #EstadoVI.Err_Protusion THEN #EstadoVI.Error_Mx := TRUE; END_IF;
END_REGION

REGION Network 59: CONTADOR SEGURIDAD PRESENCIA - CNTSeg_pHsMx
   RUNG wire#powerrail
      #CNTSeg_pHsMx(IN := wire#w3, R := wire#w6, PV := #V_CNTSeg_pHsMx, BaseUnidades_ms := "CTE_BaseUnidades_1ms", QU =>, QD =>, CVU =>, CVD =>)
   END_RUNG
   RUNG wire#powerrail
      Contact( #Mx_ET10 )
      Contact( #MEnt_DescargaAct )
      wire#w1
      Contact( #Avance_Tx )
      Contact( #Selec_M1_Entrada )
   END_RUNG wire#w3
   RUNG wire#powerrail
      Contact( #Mx_ET11 )
   END_RUNG wire#w1
   RUNG wire#powerrail
      Contact( #Mx_ET12 )
   END_RUNG wire#w1
   RUNG wire#powerrail
      Contact( #Mx_ET50 )
      wire#w2
      Contact( #Simultaneo_Mx )
      Contact( #MEnt_DescargaAct )
   END_RUNG wire#w1
   RUNG wire#powerrail
      Contact( #Mx_ET51 )
   END_RUNG wire#w2
   RUNG wire#w1
      Contact( #Retroceso_Tx )
      Contact( #Selec_M3_Entrada )
   END_RUNG wire#w3
   RUNG wire#powerrail
      I_Contact( #Mx_ET10 )
      wire#w4
      I_Contact( #Mx_ET11 )
      I_Contact( #Mx_ET12 )
      wire#w5
      I_Contact( #Mx_ET50 )
      I_Contact( #Mx_ET51 )
   END_RUNG wire#w6
   RUNG wire#powerrail
      I_Contact( #MEnt_DescargaAct )
   END_RUNG wire#w4
   RUNG wire#w5
      I_Contact( #Simultaneo_Mx )
   END_RUNG wire#w6
   RUNG wire#w5
      I_Contact( #MEnt_DescargaAct )
   END_RUNG wire#w6
   // the same network as SCL:
   #CNTSeg_pHsMx(IN := ((#Mx_ET10 AND #MEnt_DescargaAct) OR #Mx_ET11 OR #Mx_ET12 OR ((#Mx_ET50 OR #Mx_ET51) AND #Simultaneo_Mx AND #MEnt_DescargaAct)) AND ((#Avance_Tx AND #Selec_M1_Entrada) OR (#Retroceso_Tx AND #Selec_M3_Entrada)),   // "FB910_CNT_UHS"
                 R := (NOT #Mx_ET10 OR NOT #MEnt_DescargaAct) AND NOT #Mx_ET11 AND NOT #Mx_ET12 AND ((NOT #Mx_ET50 AND NOT #Mx_ET51) OR NOT #Simultaneo_Mx OR NOT #MEnt_DescargaAct),
                 PV := #V_CNTSeg_pHsMx,
                 BaseUnidades_ms := "CTE_BaseUnidades_1ms");
END_REGION

REGION Network 60: CONTADOR DE PRESENCIA - CNT_pHsMx
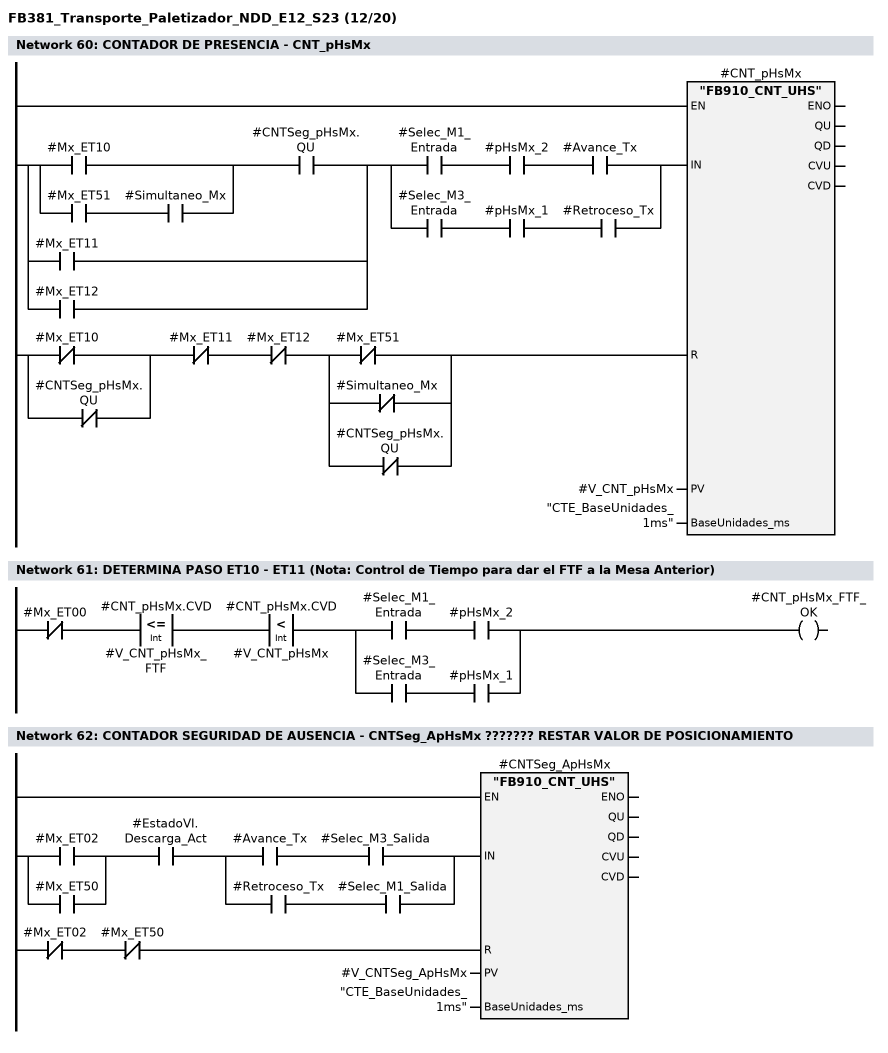
   RUNG wire#powerrail
      #CNT_pHsMx(IN := wire#w3, R := wire#w6, PV := #V_CNT_pHsMx, BaseUnidades_ms := "CTE_BaseUnidades_1ms", QU =>, QD =>, CVU =>, CVD =>)
   END_RUNG
   RUNG wire#powerrail
      Contact( #Mx_ET10 )
      wire#w1
      Contact( #CNTSeg_pHsMx.QU )
      wire#w2
      Contact( #Selec_M1_Entrada )
      Contact( #pHsMx_2 )
      Contact( #Avance_Tx )
   END_RUNG wire#w3
   RUNG wire#powerrail
      Contact( #Mx_ET51 )
      Contact( #Simultaneo_Mx )
   END_RUNG wire#w1
   RUNG wire#powerrail
      Contact( #Mx_ET11 )
   END_RUNG wire#w2
   RUNG wire#powerrail
      Contact( #Mx_ET12 )
   END_RUNG wire#w2
   RUNG wire#w2
      Contact( #Selec_M3_Entrada )
      Contact( #pHsMx_1 )
      Contact( #Retroceso_Tx )
   END_RUNG wire#w3
   RUNG wire#powerrail
      I_Contact( #Mx_ET10 )
      wire#w4
      I_Contact( #Mx_ET11 )
      I_Contact( #Mx_ET12 )
      wire#w5
      I_Contact( #Mx_ET51 )
   END_RUNG wire#w6
   RUNG wire#powerrail
      I_Contact( #CNTSeg_pHsMx.QU )
   END_RUNG wire#w4
   RUNG wire#w5
      I_Contact( #Simultaneo_Mx )
   END_RUNG wire#w6
   RUNG wire#w5
      I_Contact( #CNTSeg_pHsMx.QU )
   END_RUNG wire#w6
   // the same network as SCL:
   #CNT_pHsMx(IN := (((#Mx_ET10 OR (#Mx_ET51 AND #Simultaneo_Mx)) AND #CNTSeg_pHsMx.QU) OR #Mx_ET11 OR #Mx_ET12) AND ((#Selec_M1_Entrada AND #pHsMx_2 AND #Avance_Tx) OR (#Selec_M3_Entrada AND #pHsMx_1 AND #Retroceso_Tx)),   // "FB910_CNT_UHS"
              R := (NOT #Mx_ET10 OR NOT #CNTSeg_pHsMx.QU) AND NOT #Mx_ET11 AND NOT #Mx_ET12 AND (NOT #Mx_ET51 OR NOT #Simultaneo_Mx OR NOT #CNTSeg_pHsMx.QU),
              PV := #V_CNT_pHsMx,
              BaseUnidades_ms := "CTE_BaseUnidades_1ms");
END_REGION

REGION Network 61: DETERMINA PASO ET10 - ET11 (Nota: Control de Tiempo para dar el FTF a la Mesa Anterior)
   RUNG wire#powerrail
      I_Contact( #Mx_ET00 )
      { S7_Templates := "SrcType := Int" } LE_Contact(in1 := #CNT_pHsMx.CVD, in2 := #V_CNT_pHsMx_FTF)
      { S7_Templates := "SrcType := Int" } LT_Contact(in1 := #CNT_pHsMx.CVD, in2 := #V_CNT_pHsMx)
      wire#w1
      Contact( #Selec_M1_Entrada )
      Contact( #pHsMx_2 )
      wire#w2
      Coil( #CNT_pHsMx_FTF_OK )
   END_RUNG
   RUNG wire#w1
      Contact( #Selec_M3_Entrada )
      Contact( #pHsMx_1 )
   END_RUNG wire#w2
   // the same network as SCL:
   #CNT_pHsMx_FTF_OK := NOT #Mx_ET00 AND (#CNT_pHsMx.CVD <= #V_CNT_pHsMx_FTF) AND (#CNT_pHsMx.CVD < #V_CNT_pHsMx) AND ((#Selec_M1_Entrada AND #pHsMx_2) OR (#Selec_M3_Entrada AND #pHsMx_1));
END_REGION

REGION Network 62: CONTADOR SEGURIDAD DE AUSENCIA - CNTSeg_ApHsMx ??????? RESTAR VALOR DE POSICIONAMIENTO
   RUNG wire#powerrail
      #CNTSeg_ApHsMx(IN := wire#w3, R := wire#w4, PV := #V_CNTSeg_ApHsMx, BaseUnidades_ms := "CTE_BaseUnidades_1ms", QU =>, QD =>, CVU =>, CVD =>)
   END_RUNG
   RUNG wire#powerrail
      Contact( #Mx_ET02 )
      wire#w1
      Contact( #EstadoVI.Descarga_Act )
      wire#w2
      Contact( #Avance_Tx )
      Contact( #Selec_M3_Salida )
   END_RUNG wire#w3
   RUNG wire#powerrail
      Contact( #Mx_ET50 )
   END_RUNG wire#w1
   RUNG wire#w2
      Contact( #Retroceso_Tx )
      Contact( #Selec_M1_Salida )
   END_RUNG wire#w3
   RUNG wire#powerrail
      I_Contact( #Mx_ET02 )
      I_Contact( #Mx_ET50 )
   END_RUNG wire#w4
   // the same network as SCL:
   #CNTSeg_ApHsMx(IN := (#Mx_ET02 OR #Mx_ET50) AND #EstadoVI.Descarga_Act AND ((#Avance_Tx AND #Selec_M3_Salida) OR (#Retroceso_Tx AND #Selec_M1_Salida)),   // "FB910_CNT_UHS"
                  R := NOT #Mx_ET02 AND NOT #Mx_ET50,
                  PV := #V_CNTSeg_ApHsMx,
                  BaseUnidades_ms := "CTE_BaseUnidades_1ms");
END_REGION

REGION Network 63: CONTADOR DE LA AUSENCIA - CNT_ApHsMX
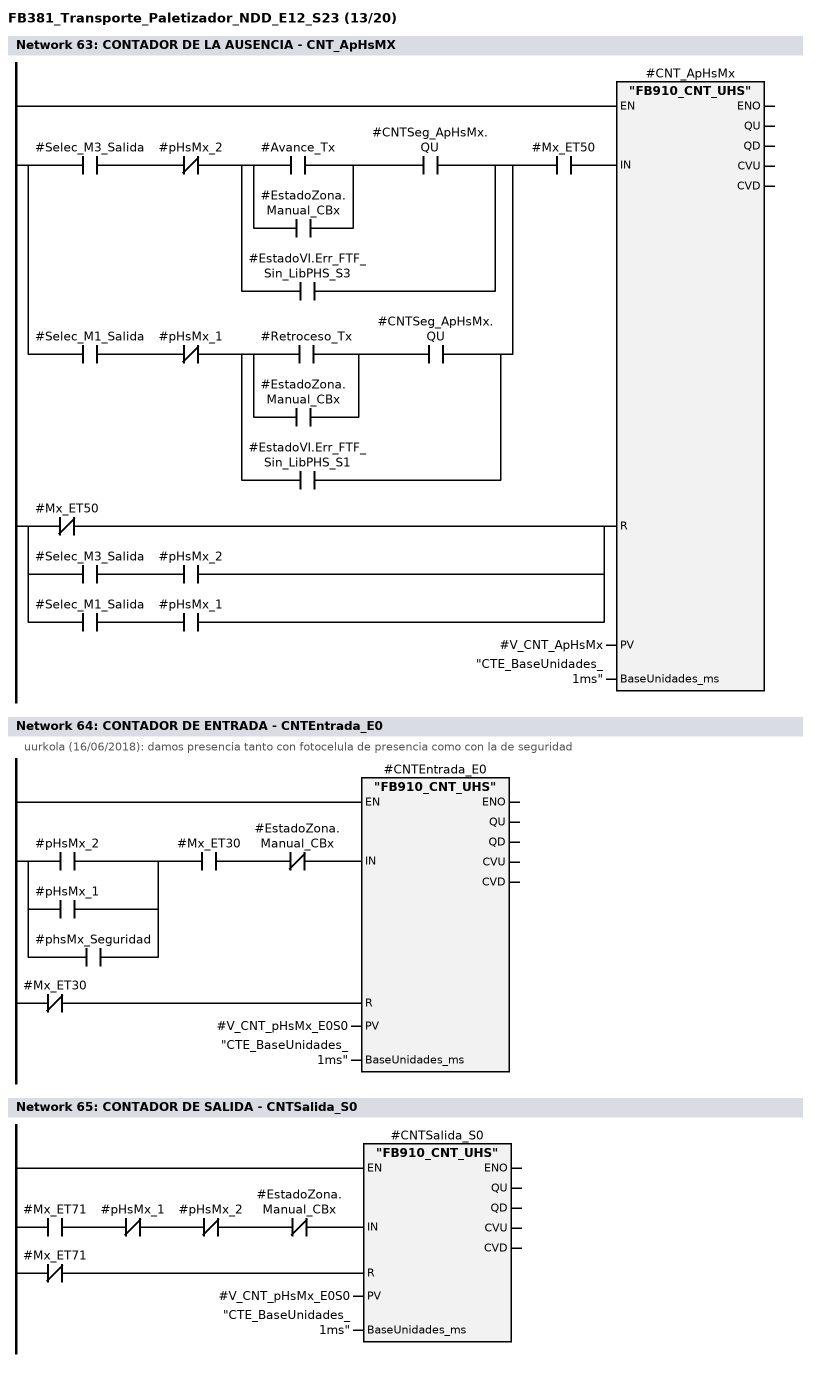
   RUNG wire#powerrail
      #CNT_ApHsMx(IN := wire#w6, R := wire#w7, PV := #V_CNT_ApHsMx, BaseUnidades_ms := "CTE_BaseUnidades_1ms", QU =>, QD =>, CVU =>, CVD =>)
   END_RUNG
   RUNG wire#powerrail
      Contact( #Selec_M3_Salida )
      I_Contact( #pHsMx_2 )
      wire#w1
      Contact( #Avance_Tx )
      wire#w2
      Contact( #CNTSeg_ApHsMx.QU )
      wire#w3
      Contact( #Mx_ET50 )
   END_RUNG wire#w6
   RUNG wire#w1
      Contact( #EstadoZona.Manual_CBx )
   END_RUNG wire#w2
   RUNG wire#w1
      Contact( #EstadoVI.Err_FTF_Sin_LibPHS_S3 )
   END_RUNG wire#w3
   RUNG wire#powerrail
      Contact( #Selec_M1_Salida )
      I_Contact( #pHsMx_1 )
      wire#w4
      Contact( #Retroceso_Tx )
      wire#w5
      Contact( #CNTSeg_ApHsMx.QU )
   END_RUNG wire#w3
   RUNG wire#w4
      Contact( #EstadoZona.Manual_CBx )
   END_RUNG wire#w5
   RUNG wire#w4
      Contact( #EstadoVI.Err_FTF_Sin_LibPHS_S1 )
   END_RUNG wire#w3
   RUNG wire#powerrail
      I_Contact( #Mx_ET50 )
   END_RUNG wire#w7
   RUNG wire#powerrail
      Contact( #Selec_M3_Salida )
      Contact( #pHsMx_2 )
   END_RUNG wire#w7
   RUNG wire#powerrail
      Contact( #Selec_M1_Salida )
      Contact( #pHsMx_1 )
   END_RUNG wire#w7
   // the same network as SCL:
   #CNT_ApHsMx(IN := ((#Selec_M3_Salida AND NOT #pHsMx_2 AND (((#Avance_Tx OR #EstadoZona.Manual_CBx) AND #CNTSeg_ApHsMx.QU) OR #EstadoVI.Err_FTF_Sin_LibPHS_S3)) OR (#Selec_M1_Salida AND NOT #pHsMx_1 AND (((#Retroceso_Tx OR #EstadoZona.Manual_CBx) AND #CNTSeg_ApHsMx.QU) OR #EstadoVI.Err_FTF_Sin_LibPHS_S1))) AND #Mx_ET50,   // "FB910_CNT_UHS"
               R := NOT #Mx_ET50 OR (#Selec_M3_Salida AND #pHsMx_2) OR (#Selec_M1_Salida AND #pHsMx_1),
               PV := #V_CNT_ApHsMx,
               BaseUnidades_ms := "CTE_BaseUnidades_1ms");
END_REGION

REGION Network 64: CONTADOR DE ENTRADA - CNTEntrada_E0
   // uurkola (16/06/2018): damos presencia tanto con fotocelula de presencia como con la de seguridad
   RUNG wire#powerrail
      #CNTEntrada_E0(IN := wire#w2, R := wire#w3, PV := #V_CNT_pHsMx_E0S0, BaseUnidades_ms := "CTE_BaseUnidades_1ms", QU =>, QD =>, CVU =>, CVD =>)
   END_RUNG
   RUNG wire#powerrail
      Contact( #pHsMx_2 )
      wire#w1
      Contact( #Mx_ET30 )
      I_Contact( #EstadoZona.Manual_CBx )
   END_RUNG wire#w2
   RUNG wire#powerrail
      Contact( #pHsMx_1 )
   END_RUNG wire#w1
   RUNG wire#powerrail
      Contact( #phsMx_Seguridad )
   END_RUNG wire#w1
   RUNG wire#powerrail
      I_Contact( #Mx_ET30 )
   END_RUNG wire#w3
   // the same network as SCL:
   #CNTEntrada_E0(IN := (#pHsMx_2 OR #pHsMx_1 OR #phsMx_Seguridad) AND #Mx_ET30 AND NOT #EstadoZona.Manual_CBx,   // "FB910_CNT_UHS"
                  R := NOT #Mx_ET30,
                  PV := #V_CNT_pHsMx_E0S0,
                  BaseUnidades_ms := "CTE_BaseUnidades_1ms");
END_REGION

REGION Network 65: CONTADOR DE SALIDA - CNTSalida_S0
   RUNG wire#powerrail
      #CNTSalida_S0(IN := wire#w1, R := wire#w2, PV := #V_CNT_pHsMx_E0S0, BaseUnidades_ms := "CTE_BaseUnidades_1ms", QU =>, QD =>, CVU =>, CVD =>)
   END_RUNG
   RUNG wire#powerrail
      Contact( #Mx_ET71 )
      I_Contact( #pHsMx_1 )
      I_Contact( #pHsMx_2 )
      I_Contact( #EstadoZona.Manual_CBx )
   END_RUNG wire#w1
   RUNG wire#powerrail
      I_Contact( #Mx_ET71 )
   END_RUNG wire#w2
   // the same network as SCL:
   #CNTSalida_S0(IN := #Mx_ET71 AND NOT #pHsMx_1 AND NOT #pHsMx_2 AND NOT #EstadoZona.Manual_CBx,   // "FB910_CNT_UHS"
                 R := NOT #Mx_ET71,
                 PV := #V_CNT_pHsMx_E0S0,
                 BaseUnidades_ms := "CTE_BaseUnidades_1ms");
END_REGION

REGION Network 66: VARIABLES AUXILIARES - Fin de Reset
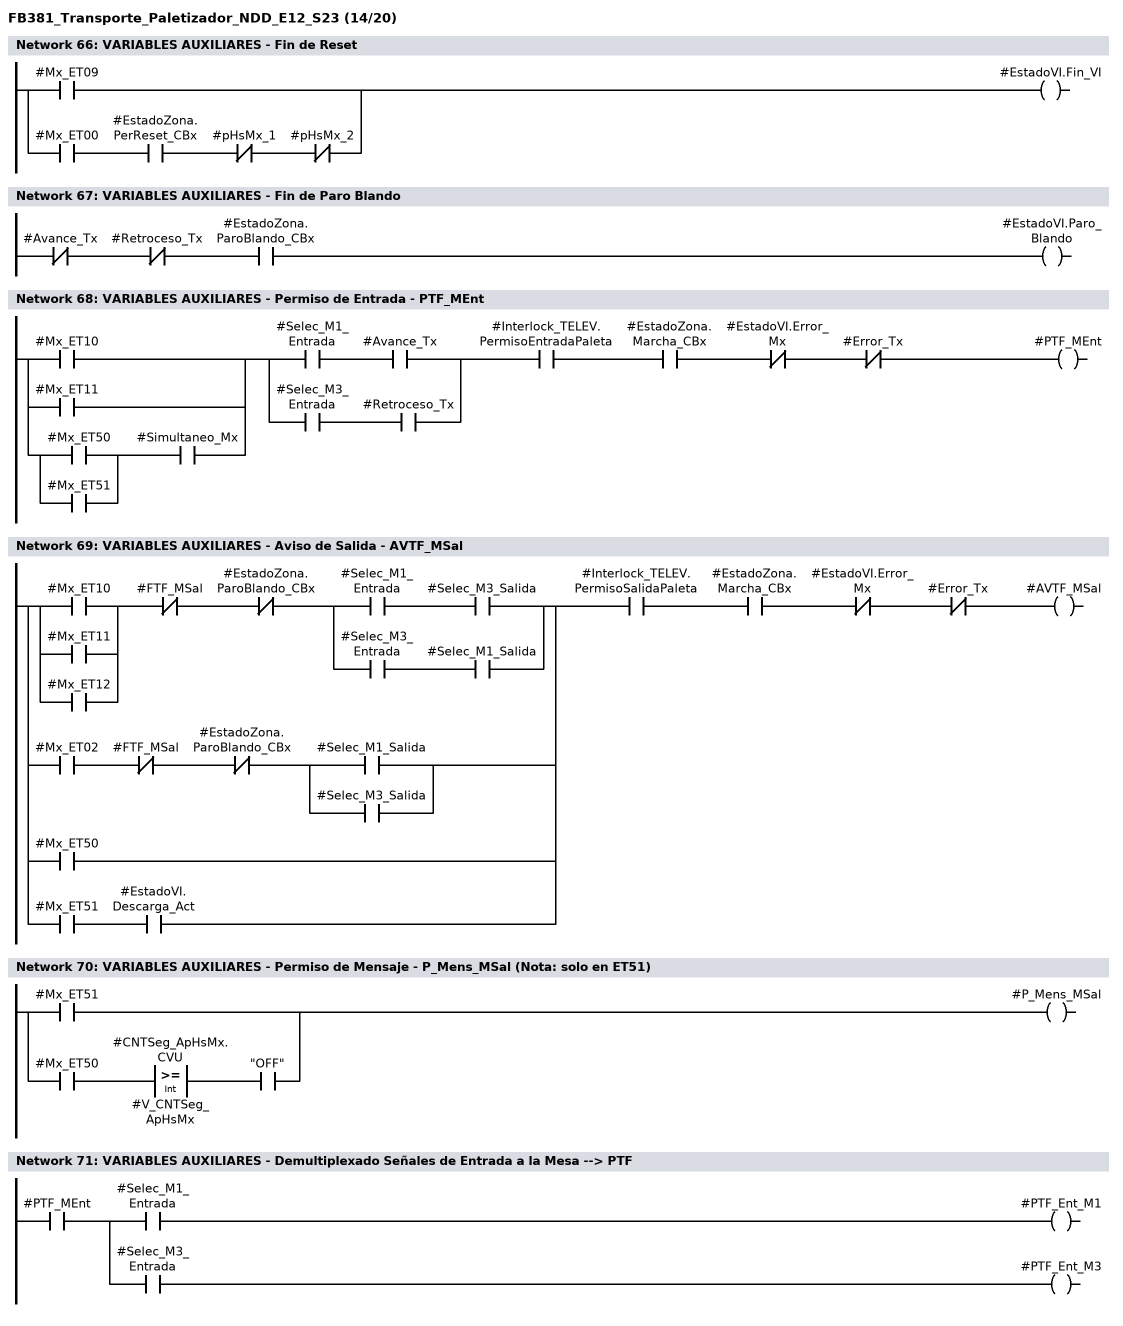
   RUNG wire#powerrail
      Contact( #Mx_ET09 )
      wire#w1
      Coil( #EstadoVI.Fin_VI )
   END_RUNG
   RUNG wire#powerrail
      Contact( #Mx_ET00 )
      Contact( #EstadoZona.PerReset_CBx )
      I_Contact( #pHsMx_1 )
      I_Contact( #pHsMx_2 )
   END_RUNG wire#w1
   // the same network as SCL:
   #EstadoVI.Fin_VI := #Mx_ET09 OR (#Mx_ET00 AND #EstadoZona.PerReset_CBx AND NOT #pHsMx_1 AND NOT #pHsMx_2);
END_REGION

REGION Network 67: VARIABLES AUXILIARES - Fin de Paro Blando
   RUNG wire#powerrail
      I_Contact( #Avance_Tx )
      I_Contact( #Retroceso_Tx )
      Contact( #EstadoZona.ParoBlando_CBx )
      Coil( #EstadoVI.Paro_Blando )
   END_RUNG
   // the same network as SCL:
   #EstadoVI.Paro_Blando := NOT #Avance_Tx AND NOT #Retroceso_Tx AND #EstadoZona.ParoBlando_CBx;
END_REGION

REGION Network 68: VARIABLES AUXILIARES - Permiso de Entrada - PTF_MEnt
   RUNG wire#powerrail
      Contact( #Mx_ET10 )
      wire#w1
      Contact( #Selec_M1_Entrada )
      Contact( #Avance_Tx )
      wire#w3
      Contact( #Interlock_TELEV.PermisoEntradaPaleta )
      Contact( #EstadoZona.Marcha_CBx )
      I_Contact( #EstadoVI.Error_Mx )
      I_Contact( #Error_Tx )
      Coil( #PTF_MEnt )
   END_RUNG
   RUNG wire#powerrail
      Contact( #Mx_ET11 )
   END_RUNG wire#w1
   RUNG wire#powerrail
      Contact( #Mx_ET50 )
      wire#w2
      Contact( #Simultaneo_Mx )
   END_RUNG wire#w1
   RUNG wire#powerrail
      Contact( #Mx_ET51 )
   END_RUNG wire#w2
   RUNG wire#w1
      Contact( #Selec_M3_Entrada )
      Contact( #Retroceso_Tx )
   END_RUNG wire#w3
   // the same network as SCL:
   #PTF_MEnt := (#Mx_ET10 OR #Mx_ET11 OR ((#Mx_ET50 OR #Mx_ET51) AND #Simultaneo_Mx)) AND ((#Selec_M1_Entrada AND #Avance_Tx) OR (#Selec_M3_Entrada AND #Retroceso_Tx)) AND #Interlock_TELEV.PermisoEntradaPaleta AND #EstadoZona.Marcha_CBx AND NOT #EstadoVI.Error_Mx AND NOT #Error_Tx;
END_REGION

REGION Network 69: VARIABLES AUXILIARES - Aviso de Salida - AVTF_MSal
   RUNG wire#powerrail
      Contact( #Mx_ET10 )
      wire#w1
      I_Contact( #FTF_MSal )
      I_Contact( #EstadoZona.ParoBlando_CBx )
      wire#w2
      Contact( #Selec_M1_Entrada )
      Contact( #Selec_M3_Salida )
      wire#w3
      Contact( #Interlock_TELEV.PermisoSalidaPaleta )
      Contact( #EstadoZona.Marcha_CBx )
      I_Contact( #EstadoVI.Error_Mx )
      I_Contact( #Error_Tx )
      Coil( #AVTF_MSal )
   END_RUNG
   RUNG wire#powerrail
      Contact( #Mx_ET11 )
   END_RUNG wire#w1
   RUNG wire#powerrail
      Contact( #Mx_ET12 )
   END_RUNG wire#w1
   RUNG wire#w2
      Contact( #Selec_M3_Entrada )
      Contact( #Selec_M1_Salida )
   END_RUNG wire#w3
   RUNG wire#powerrail
      Contact( #Mx_ET02 )
      I_Contact( #FTF_MSal )
      I_Contact( #EstadoZona.ParoBlando_CBx )
      wire#w4
      Contact( #Selec_M1_Salida )
   END_RUNG wire#w3
   RUNG wire#w4
      Contact( #Selec_M3_Salida )
   END_RUNG wire#w3
   RUNG wire#powerrail
      Contact( #Mx_ET50 )
   END_RUNG wire#w3
   RUNG wire#powerrail
      Contact( #Mx_ET51 )
      Contact( #EstadoVI.Descarga_Act )
   END_RUNG wire#w3
   // the same network as SCL:
   #AVTF_MSal := (((#Mx_ET10 OR #Mx_ET11 OR #Mx_ET12) AND NOT #FTF_MSal AND NOT #EstadoZona.ParoBlando_CBx AND ((#Selec_M1_Entrada AND #Selec_M3_Salida) OR (#Selec_M3_Entrada AND #Selec_M1_Salida))) OR (#Mx_ET02 AND NOT #FTF_MSal AND NOT #EstadoZona.ParoBlando_CBx AND (#Selec_M1_Salida OR #Selec_M3_Salida)) OR #Mx_ET50 OR (#Mx_ET51 AND #EstadoVI.Descarga_Act)) AND #Interlock_TELEV.PermisoSalidaPaleta AND #EstadoZona.Marcha_CBx AND NOT #EstadoVI.Error_Mx AND NOT #Error_Tx;
END_REGION

REGION Network 70: VARIABLES AUXILIARES - Permiso de Mensaje - P_Mens_MSal (Nota: solo en ET51)
   RUNG wire#powerrail
      Contact( #Mx_ET51 )
      wire#w1
      Coil( #P_Mens_MSal )
   END_RUNG
   RUNG wire#powerrail
      Contact( #Mx_ET50 )
      { S7_Templates := "SrcType := Int" } GE_Contact(in1 := #CNTSeg_ApHsMx.CVU, in2 := #V_CNTSeg_ApHsMx)
      Contact( "OFF" )
   END_RUNG wire#w1
   // the same network as SCL:
   #P_Mens_MSal := #Mx_ET51 OR (#Mx_ET50 AND (#CNTSeg_ApHsMx.CVU >= #V_CNTSeg_ApHsMx) AND "OFF");
END_REGION

REGION Network 71: VARIABLES AUXILIARES - Demultiplexado Señales de Entrada a la Mesa --> PTF
   RUNG wire#powerrail
      Contact( #PTF_MEnt )
      wire#w1
      Contact( #Selec_M1_Entrada )
      Coil( #PTF_Ent_M1 )
   END_RUNG
   RUNG wire#w1
      Contact( #Selec_M3_Entrada )
      Coil( #PTF_Ent_M3 )
   END_RUNG
   // the same network as SCL:
   #PTF_Ent_M1 := #PTF_MEnt AND #Selec_M1_Entrada;
   #PTF_Ent_M3 := #PTF_MEnt AND #Selec_M3_Entrada;
END_REGION

REGION Network 72: VARIABLES AUXILIARES - Demultiplexado Señales de Entrada a la Mesa --> FTF
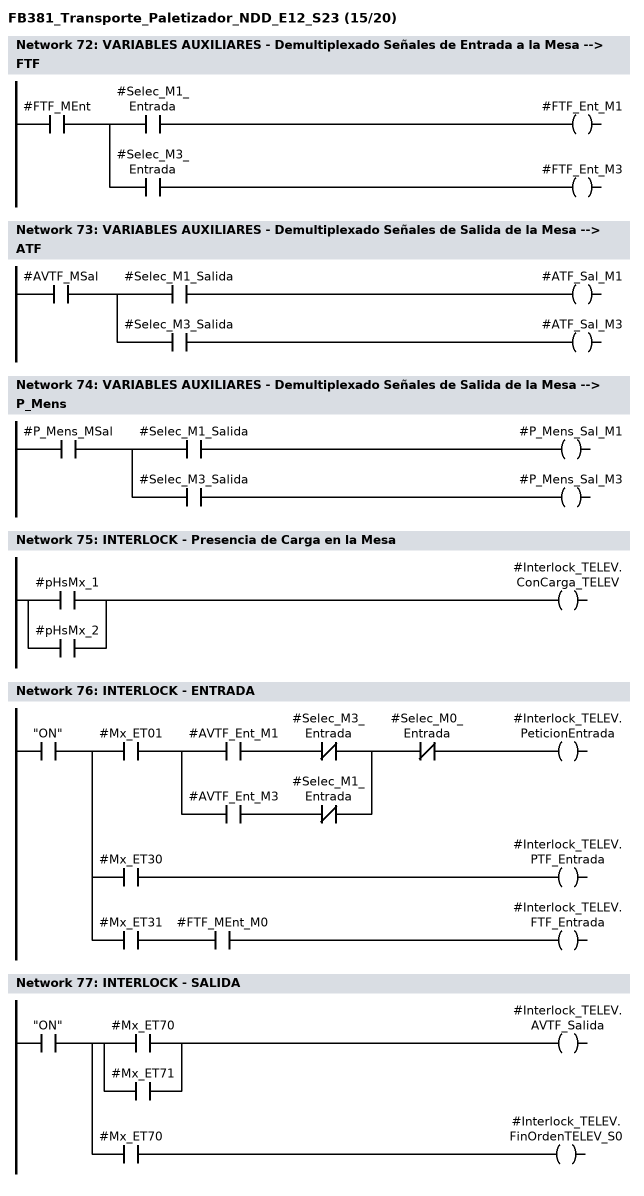
   RUNG wire#powerrail
      Contact( #FTF_MEnt )
      wire#w1
      Contact( #Selec_M1_Entrada )
      Coil( #FTF_Ent_M1 )
   END_RUNG
   RUNG wire#w1
      Contact( #Selec_M3_Entrada )
      Coil( #FTF_Ent_M3 )
   END_RUNG
   // the same network as SCL:
   #FTF_Ent_M1 := #FTF_MEnt AND #Selec_M1_Entrada;
   #FTF_Ent_M3 := #FTF_MEnt AND #Selec_M3_Entrada;
END_REGION

REGION Network 73: VARIABLES AUXILIARES - Demultiplexado Señales de Salida de la Mesa --> ATF
   RUNG wire#powerrail
      Contact( #AVTF_MSal )
      wire#w1
      Contact( #Selec_M1_Salida )
      Coil( #ATF_Sal_M1 )
   END_RUNG
   RUNG wire#w1
      Contact( #Selec_M3_Salida )
      Coil( #ATF_Sal_M3 )
   END_RUNG
   // the same network as SCL:
   #ATF_Sal_M1 := #AVTF_MSal AND #Selec_M1_Salida;
   #ATF_Sal_M3 := #AVTF_MSal AND #Selec_M3_Salida;
END_REGION

REGION Network 74: VARIABLES AUXILIARES - Demultiplexado Señales de Salida de la Mesa --> P_Mens
   RUNG wire#powerrail
      Contact( #P_Mens_MSal )
      wire#w1
      Contact( #Selec_M1_Salida )
      Coil( #P_Mens_Sal_M1 )
   END_RUNG
   RUNG wire#w1
      Contact( #Selec_M3_Salida )
      Coil( #P_Mens_Sal_M3 )
   END_RUNG
   // the same network as SCL:
   #P_Mens_Sal_M1 := #P_Mens_MSal AND #Selec_M1_Salida;
   #P_Mens_Sal_M3 := #P_Mens_MSal AND #Selec_M3_Salida;
END_REGION

REGION Network 75: INTERLOCK - Presencia de Carga en la Mesa
   RUNG wire#powerrail
      Contact( #pHsMx_1 )
      wire#w1
      Coil( #Interlock_TELEV.ConCarga_TELEV )
   END_RUNG
   RUNG wire#powerrail
      Contact( #pHsMx_2 )
   END_RUNG wire#w1
   // the same network as SCL:
   #Interlock_TELEV.ConCarga_TELEV := #pHsMx_1 OR #pHsMx_2;
END_REGION

REGION Network 76: INTERLOCK - ENTRADA
   RUNG wire#powerrail
      Contact( "ON" )
      wire#w1
      Contact( #Mx_ET01 )
      wire#w2
      Contact( #AVTF_Ent_M1 )
      I_Contact( #Selec_M3_Entrada )
      wire#w3
      I_Contact( #Selec_M0_Entrada )
      Coil( #Interlock_TELEV.PeticionEntrada )
   END_RUNG
   RUNG wire#w2
      Contact( #AVTF_Ent_M3 )
      I_Contact( #Selec_M1_Entrada )
   END_RUNG wire#w3
   RUNG wire#w1
      Contact( #Mx_ET30 )
      Coil( #Interlock_TELEV.PTF_Entrada )
   END_RUNG
   RUNG wire#w1
      Contact( #Mx_ET31 )
      Contact( #FTF_MEnt_M0 )
      Coil( #Interlock_TELEV.FTF_Entrada )
   END_RUNG
   // the same network as SCL:
   #Interlock_TELEV.PeticionEntrada := "ON" AND #Mx_ET01 AND ((#AVTF_Ent_M1 AND NOT #Selec_M3_Entrada) OR (#AVTF_Ent_M3 AND NOT #Selec_M1_Entrada)) AND NOT #Selec_M0_Entrada;
   #Interlock_TELEV.PTF_Entrada := "ON" AND #Mx_ET30;
   #Interlock_TELEV.FTF_Entrada := "ON" AND #Mx_ET31 AND #FTF_MEnt_M0;
END_REGION

REGION Network 77: INTERLOCK - SALIDA
   RUNG wire#powerrail
      Contact( "ON" )
      wire#w1
      Contact( #Mx_ET70 )
      wire#w2
      Coil( #Interlock_TELEV.AVTF_Salida )
   END_RUNG
   RUNG wire#w1
      Contact( #Mx_ET71 )
   END_RUNG wire#w2
   RUNG wire#w1
      Contact( #Mx_ET70 )
      Coil( #Interlock_TELEV.FinOrdenTELEV_S0 )
   END_RUNG
   // the same network as SCL:
   #Interlock_TELEV.AVTF_Salida := "ON" AND (#Mx_ET70 OR #Mx_ET71);
   #Interlock_TELEV.FinOrdenTELEV_S0 := "ON" AND #Mx_ET70;
END_REGION

REGION Network 78: CONTADOR DE SIMULTANEO
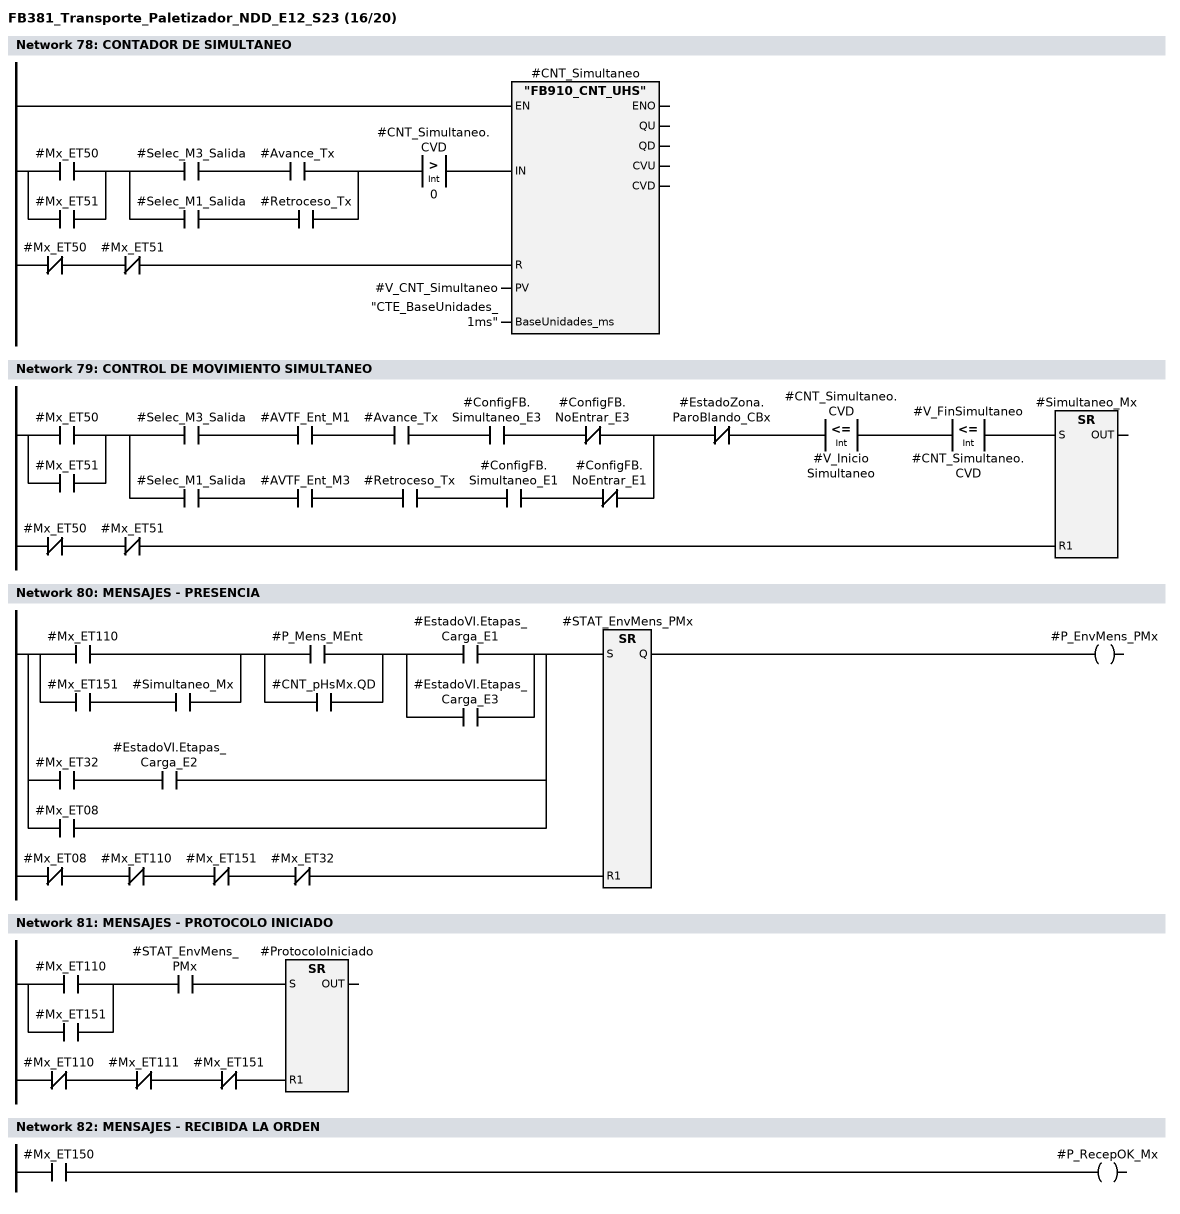
   RUNG wire#powerrail
      #CNT_Simultaneo(IN := wire#w3, R := wire#w4, PV := #V_CNT_Simultaneo, BaseUnidades_ms := "CTE_BaseUnidades_1ms", QU =>, QD =>, CVU =>, CVD =>)
   END_RUNG
   RUNG wire#powerrail
      Contact( #Mx_ET50 )
      wire#w1
      Contact( #Selec_M3_Salida )
      Contact( #Avance_Tx )
      wire#w2
      { S7_Templates := "SrcType := Int" } GT_Contact(in1 := #CNT_Simultaneo.CVD, in2 := 0)
   END_RUNG wire#w3
   RUNG wire#powerrail
      Contact( #Mx_ET51 )
   END_RUNG wire#w1
   RUNG wire#w1
      Contact( #Selec_M1_Salida )
      Contact( #Retroceso_Tx )
   END_RUNG wire#w2
   RUNG wire#powerrail
      I_Contact( #Mx_ET50 )
      I_Contact( #Mx_ET51 )
   END_RUNG wire#w4
   // the same network as SCL:
   #CNT_Simultaneo(IN := (#Mx_ET50 OR #Mx_ET51) AND ((#Selec_M3_Salida AND #Avance_Tx) OR (#Selec_M1_Salida AND #Retroceso_Tx)) AND (#CNT_Simultaneo.CVD > 0),   // "FB910_CNT_UHS"
                   R := NOT #Mx_ET50 AND NOT #Mx_ET51,
                   PV := #V_CNT_Simultaneo,
                   BaseUnidades_ms := "CTE_BaseUnidades_1ms");
END_REGION

REGION Network 79: CONTROL DE MOVIMIENTO SIMULTANEO
   RUNG wire#powerrail
      Contact( #Mx_ET50 )
      wire#w1
      Contact( #Selec_M3_Salida )
      Contact( #AVTF_Ent_M1 )
      Contact( #Avance_Tx )
      Contact( #ConfigFB.Simultaneo_E3 )
      I_Contact( #ConfigFB.NoEntrar_E3 )
      wire#w2
      I_Contact( #EstadoZona.ParoBlando_CBx )
      { S7_Templates := "SrcType := Int" } LE_Contact(in1 := #CNT_Simultaneo.CVD, in2 := #V_InicioSimultaneo)
      { S7_Templates := "SrcType := Int" } LE_Contact(in1 := #V_FinSimultaneo, in2 := #CNT_Simultaneo.CVD)
      S_SR(operand := #Simultaneo_Mx, r1 := wire#w3)
   END_RUNG
   RUNG wire#powerrail
      Contact( #Mx_ET51 )
   END_RUNG wire#w1
   RUNG wire#w1
      Contact( #Selec_M1_Salida )
      Contact( #AVTF_Ent_M3 )
      Contact( #Retroceso_Tx )
      Contact( #ConfigFB.Simultaneo_E1 )
      I_Contact( #ConfigFB.NoEntrar_E1 )
   END_RUNG wire#w2
   RUNG wire#powerrail
      I_Contact( #Mx_ET50 )
      I_Contact( #Mx_ET51 )
   END_RUNG wire#w3
   // the same network as SCL:
   IF (#Mx_ET50 OR #Mx_ET51) AND ((#Selec_M3_Salida AND #AVTF_Ent_M1 AND #Avance_Tx AND #ConfigFB.Simultaneo_E3 AND NOT #ConfigFB.NoEntrar_E3) OR (#Selec_M1_Salida AND #AVTF_Ent_M3 AND #Retroceso_Tx AND #ConfigFB.Simultaneo_E1 AND NOT #ConfigFB.NoEntrar_E1)) AND NOT #EstadoZona.ParoBlando_CBx AND (#CNT_Simultaneo.CVD <= #V_InicioSimultaneo) AND (#V_FinSimultaneo <= #CNT_Simultaneo.CVD) THEN
       #Simultaneo_Mx := TRUE;   // SR flip-flop
   END_IF;
   IF NOT #Mx_ET50 AND NOT #Mx_ET51 THEN #Simultaneo_Mx := FALSE; END_IF;
END_REGION

REGION Network 80: MENSAJES - PRESENCIA
   RUNG wire#powerrail
      Contact( #Mx_ET110 )
      wire#w1
      Contact( #P_Mens_MEnt )
      wire#w2
      Contact( #EstadoVI.Etapas_Carga_E1 )
      wire#w3
      S_SR(operand := #STAT_EnvMens_PMx, r1 := wire#w4)
      Coil( #P_EnvMens_PMx )
   END_RUNG
   RUNG wire#powerrail
      Contact( #Mx_ET151 )
      Contact( #Simultaneo_Mx )
   END_RUNG wire#w1
   RUNG wire#w1
      Contact( #CNT_pHsMx.QD )
   END_RUNG wire#w2
   RUNG wire#w2
      Contact( #EstadoVI.Etapas_Carga_E3 )
   END_RUNG wire#w3
   RUNG wire#powerrail
      Contact( #Mx_ET32 )
      Contact( #EstadoVI.Etapas_Carga_E2 )
   END_RUNG wire#w3
   RUNG wire#powerrail
      Contact( #Mx_ET08 )
   END_RUNG wire#w3
   RUNG wire#powerrail
      I_Contact( #Mx_ET08 )
      I_Contact( #Mx_ET110 )
      I_Contact( #Mx_ET151 )
      I_Contact( #Mx_ET32 )
   END_RUNG wire#w4
   // the same network as SCL:
   IF ((#Mx_ET110 OR (#Mx_ET151 AND #Simultaneo_Mx)) AND (#P_Mens_MEnt OR #CNT_pHsMx.QD) AND (#EstadoVI.Etapas_Carga_E1 OR #EstadoVI.Etapas_Carga_E3)) OR (#Mx_ET32 AND #EstadoVI.Etapas_Carga_E2) OR #Mx_ET08 THEN
       #STAT_EnvMens_PMx := TRUE;   // SR flip-flop
   END_IF;
   IF NOT #Mx_ET08 AND NOT #Mx_ET110 AND NOT #Mx_ET151 AND NOT #Mx_ET32 THEN
       #STAT_EnvMens_PMx := FALSE;
   END_IF;
   #P_EnvMens_PMx := #STAT_EnvMens_PMx;
END_REGION

REGION Network 81: MENSAJES - PROTOCOLO INICIADO
   RUNG wire#powerrail
      Contact( #Mx_ET110 )
      wire#w1
      Contact( #STAT_EnvMens_PMx )
      S_SR(operand := #ProtocoloIniciado, r1 := wire#w2)
   END_RUNG
   RUNG wire#powerrail
      Contact( #Mx_ET151 )
   END_RUNG wire#w1
   RUNG wire#powerrail
      I_Contact( #Mx_ET110 )
      I_Contact( #Mx_ET111 )
      I_Contact( #Mx_ET151 )
   END_RUNG wire#w2
   // the same network as SCL:
   IF (#Mx_ET110 OR #Mx_ET151) AND #STAT_EnvMens_PMx THEN
       #ProtocoloIniciado := TRUE;   // SR flip-flop
   END_IF;
   IF NOT #Mx_ET110 AND NOT #Mx_ET111 AND NOT #Mx_ET151 THEN #ProtocoloIniciado := FALSE; END_IF;
END_REGION

REGION Network 82: MENSAJES - RECIBIDA LA ORDEN
   RUNG wire#powerrail
      Contact( #Mx_ET150 )
      Coil( #P_RecepOK_Mx )
   END_RUNG
   // the same network as SCL:
   #P_RecepOK_Mx := #Mx_ET150;
END_REGION

REGION Network 83: SALIDAS - Avance E1E3
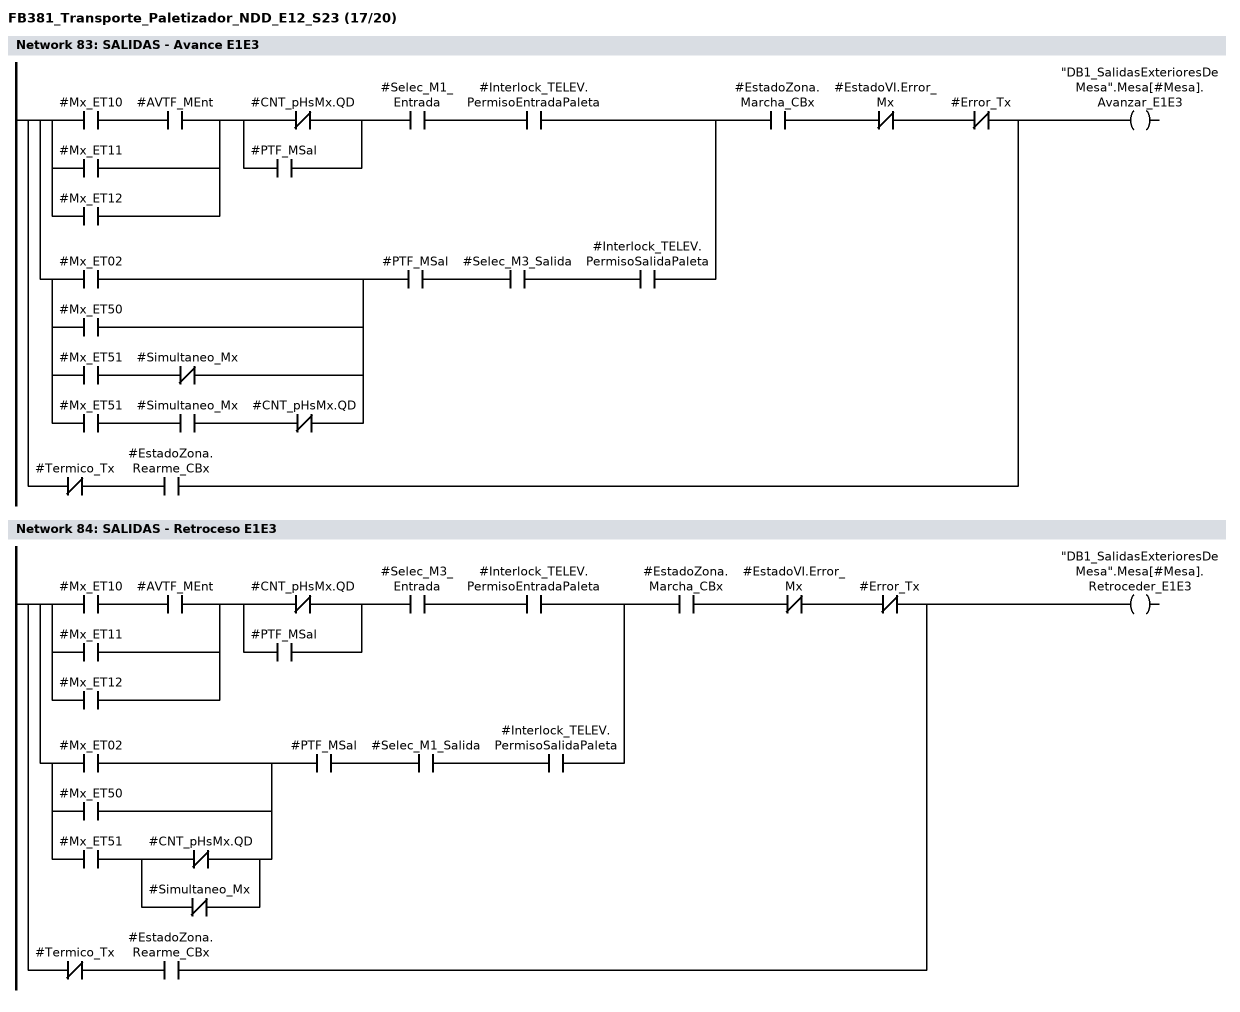
   RUNG wire#powerrail
      Contact( #Mx_ET10 )
      Contact( #AVTF_MEnt )
      wire#w1
      I_Contact( #CNT_pHsMx.QD )
      wire#w2
      Contact( #Selec_M1_Entrada )
      Contact( #Interlock_TELEV.PermisoEntradaPaleta )
      wire#w3
      Contact( #EstadoZona.Marcha_CBx )
      I_Contact( #EstadoVI.Error_Mx )
      I_Contact( #Error_Tx )
      wire#w5
      Coil( "DB1_SalidasExterioresDeMesa".Mesa[#Mesa].Avanzar_E1E3 )
   END_RUNG
   RUNG wire#powerrail
      Contact( #Mx_ET11 )
   END_RUNG wire#w1
   RUNG wire#powerrail
      Contact( #Mx_ET12 )
   END_RUNG wire#w1
   RUNG wire#w1
      Contact( #PTF_MSal )
   END_RUNG wire#w2
   RUNG wire#powerrail
      Contact( #Mx_ET02 )
      wire#w4
      Contact( #PTF_MSal )
      Contact( #Selec_M3_Salida )
      Contact( #Interlock_TELEV.PermisoSalidaPaleta )
   END_RUNG wire#w3
   RUNG wire#powerrail
      Contact( #Mx_ET50 )
   END_RUNG wire#w4
   RUNG wire#powerrail
      Contact( #Mx_ET51 )
      I_Contact( #Simultaneo_Mx )
   END_RUNG wire#w4
   RUNG wire#powerrail
      Contact( #Mx_ET51 )
      Contact( #Simultaneo_Mx )
      I_Contact( #CNT_pHsMx.QD )
   END_RUNG wire#w4
   RUNG wire#powerrail
      I_Contact( #Termico_Tx )
      Contact( #EstadoZona.Rearme_CBx )
   END_RUNG wire#w5
   // the same network as SCL:
   "DB1_SalidasExterioresDeMesa".Mesa[#Mesa].Avanzar_E1E3 := (((((#Mx_ET10 AND #AVTF_MEnt) OR #Mx_ET11 OR #Mx_ET12) AND (NOT #CNT_pHsMx.QD OR #PTF_MSal) AND #Selec_M1_Entrada AND #Interlock_TELEV.PermisoEntradaPaleta) OR ((#Mx_ET02 OR #Mx_ET50 OR (#Mx_ET51 AND NOT #Simultaneo_Mx) OR (#Mx_ET51 AND #Simultaneo_Mx AND NOT #CNT_pHsMx.QD)) AND #PTF_MSal AND #Selec_M3_Salida AND #Interlock_TELEV.PermisoSalidaPaleta)) AND #EstadoZona.Marcha_CBx AND NOT #EstadoVI.Error_Mx AND NOT #Error_Tx) OR (NOT #Termico_Tx AND #EstadoZona.Rearme_CBx);
END_REGION

REGION Network 84: SALIDAS - Retroceso E1E3
   RUNG wire#powerrail
      Contact( #Mx_ET10 )
      Contact( #AVTF_MEnt )
      wire#w1
      I_Contact( #CNT_pHsMx.QD )
      wire#w2
      Contact( #Selec_M3_Entrada )
      Contact( #Interlock_TELEV.PermisoEntradaPaleta )
      wire#w3
      Contact( #EstadoZona.Marcha_CBx )
      I_Contact( #EstadoVI.Error_Mx )
      I_Contact( #Error_Tx )
      wire#w6
      Coil( "DB1_SalidasExterioresDeMesa".Mesa[#Mesa].Retroceder_E1E3 )
   END_RUNG
   RUNG wire#powerrail
      Contact( #Mx_ET11 )
   END_RUNG wire#w1
   RUNG wire#powerrail
      Contact( #Mx_ET12 )
   END_RUNG wire#w1
   RUNG wire#w1
      Contact( #PTF_MSal )
   END_RUNG wire#w2
   RUNG wire#powerrail
      Contact( #Mx_ET02 )
      wire#w4
      Contact( #PTF_MSal )
      Contact( #Selec_M1_Salida )
      Contact( #Interlock_TELEV.PermisoSalidaPaleta )
   END_RUNG wire#w3
   RUNG wire#powerrail
      Contact( #Mx_ET50 )
   END_RUNG wire#w4
   RUNG wire#powerrail
      Contact( #Mx_ET51 )
      wire#w5
      I_Contact( #CNT_pHsMx.QD )
   END_RUNG wire#w4
   RUNG wire#w5
      I_Contact( #Simultaneo_Mx )
   END_RUNG wire#w4
   RUNG wire#powerrail
      I_Contact( #Termico_Tx )
      Contact( #EstadoZona.Rearme_CBx )
   END_RUNG wire#w6
   // the same network as SCL:
   "DB1_SalidasExterioresDeMesa".Mesa[#Mesa].Retroceder_E1E3 := (((((#Mx_ET10 AND #AVTF_MEnt) OR #Mx_ET11 OR #Mx_ET12) AND (NOT #CNT_pHsMx.QD OR #PTF_MSal) AND #Selec_M3_Entrada AND #Interlock_TELEV.PermisoEntradaPaleta) OR ((#Mx_ET02 OR #Mx_ET50 OR (#Mx_ET51 AND (NOT #CNT_pHsMx.QD OR NOT #Simultaneo_Mx))) AND #PTF_MSal AND #Selec_M1_Salida AND #Interlock_TELEV.PermisoSalidaPaleta)) AND #EstadoZona.Marcha_CBx AND NOT #EstadoVI.Error_Mx AND NOT #Error_Tx) OR (NOT #Termico_Tx AND #EstadoZona.Rearme_CBx);
END_REGION

REGION Network 85: SALIDAS - Parar E1E3
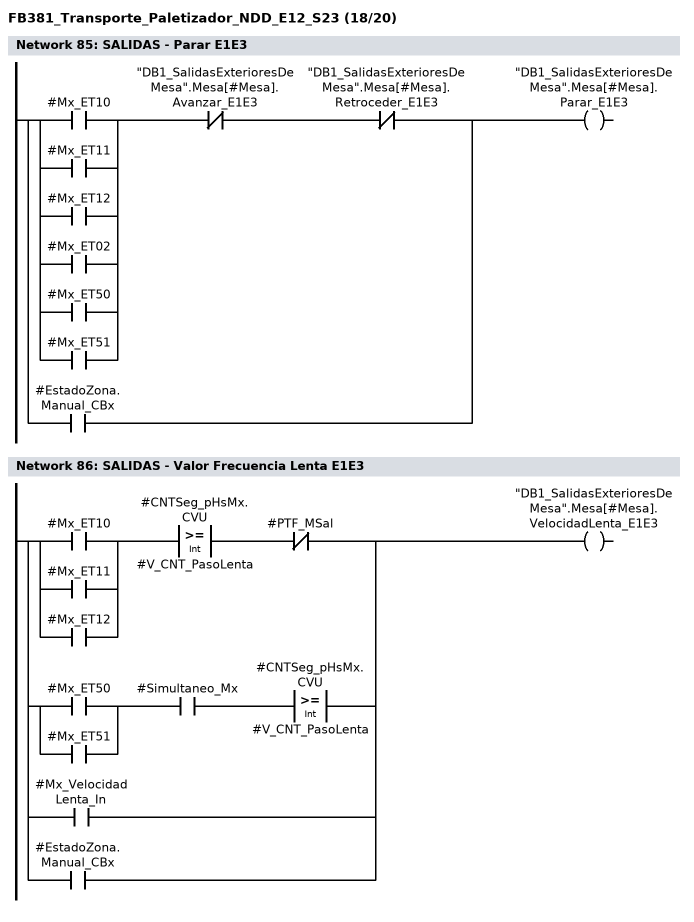
   RUNG wire#powerrail
      Contact( #Mx_ET10 )
      wire#w1
      I_Contact( "DB1_SalidasExterioresDeMesa".Mesa[#Mesa].Avanzar_E1E3 )
      I_Contact( "DB1_SalidasExterioresDeMesa".Mesa[#Mesa].Retroceder_E1E3 )
      wire#w2
      Coil( "DB1_SalidasExterioresDeMesa".Mesa[#Mesa].Parar_E1E3 )
   END_RUNG
   RUNG wire#powerrail
      Contact( #Mx_ET11 )
   END_RUNG wire#w1
   RUNG wire#powerrail
      Contact( #Mx_ET12 )
   END_RUNG wire#w1
   RUNG wire#powerrail
      Contact( #Mx_ET02 )
   END_RUNG wire#w1
   RUNG wire#powerrail
      Contact( #Mx_ET50 )
   END_RUNG wire#w1
   RUNG wire#powerrail
      Contact( #Mx_ET51 )
   END_RUNG wire#w1
   RUNG wire#powerrail
      Contact( #EstadoZona.Manual_CBx )
   END_RUNG wire#w2
   // the same network as SCL:
   "DB1_SalidasExterioresDeMesa".Mesa[#Mesa].Parar_E1E3 := ((#Mx_ET10 OR #Mx_ET11 OR #Mx_ET12 OR #Mx_ET02 OR #Mx_ET50 OR #Mx_ET51) AND NOT "DB1_SalidasExterioresDeMesa".Mesa[#Mesa].Avanzar_E1E3 AND NOT "DB1_SalidasExterioresDeMesa".Mesa[#Mesa].Retroceder_E1E3) OR #EstadoZona.Manual_CBx;
END_REGION

REGION Network 86: SALIDAS - Valor Frecuencia Lenta E1E3
   RUNG wire#powerrail
      Contact( #Mx_ET10 )
      wire#w1
      { S7_Templates := "SrcType := Int" } GE_Contact(in1 := #CNTSeg_pHsMx.CVU, in2 := #V_CNT_PasoLenta)
      I_Contact( #PTF_MSal )
      wire#w2
      Coil( "DB1_SalidasExterioresDeMesa".Mesa[#Mesa].VelocidadLenta_E1E3 )
   END_RUNG
   RUNG wire#powerrail
      Contact( #Mx_ET11 )
   END_RUNG wire#w1
   RUNG wire#powerrail
      Contact( #Mx_ET12 )
   END_RUNG wire#w1
   RUNG wire#powerrail
      Contact( #Mx_ET50 )
      wire#w3
      Contact( #Simultaneo_Mx )
      { S7_Templates := "SrcType := Int" } GE_Contact(in1 := #CNTSeg_pHsMx.CVU, in2 := #V_CNT_PasoLenta)
   END_RUNG wire#w2
   RUNG wire#powerrail
      Contact( #Mx_ET51 )
   END_RUNG wire#w3
   RUNG wire#powerrail
      Contact( #Mx_VelocidadLenta_In )
   END_RUNG wire#w2
   RUNG wire#powerrail
      Contact( #EstadoZona.Manual_CBx )
   END_RUNG wire#w2
   // the same network as SCL:
   "DB1_SalidasExterioresDeMesa".Mesa[#Mesa].VelocidadLenta_E1E3 := ((#Mx_ET10 OR #Mx_ET11 OR #Mx_ET12) AND (#CNTSeg_pHsMx.CVU >= #V_CNT_PasoLenta) AND NOT #PTF_MSal) OR ((#Mx_ET50 OR #Mx_ET51) AND #Simultaneo_Mx AND (#CNTSeg_pHsMx.CVU >= #V_CNT_PasoLenta)) OR #Mx_VelocidadLenta_In OR #EstadoZona.Manual_CBx;
END_REGION

REGION Network 87: ESTADOS DE LA MESA
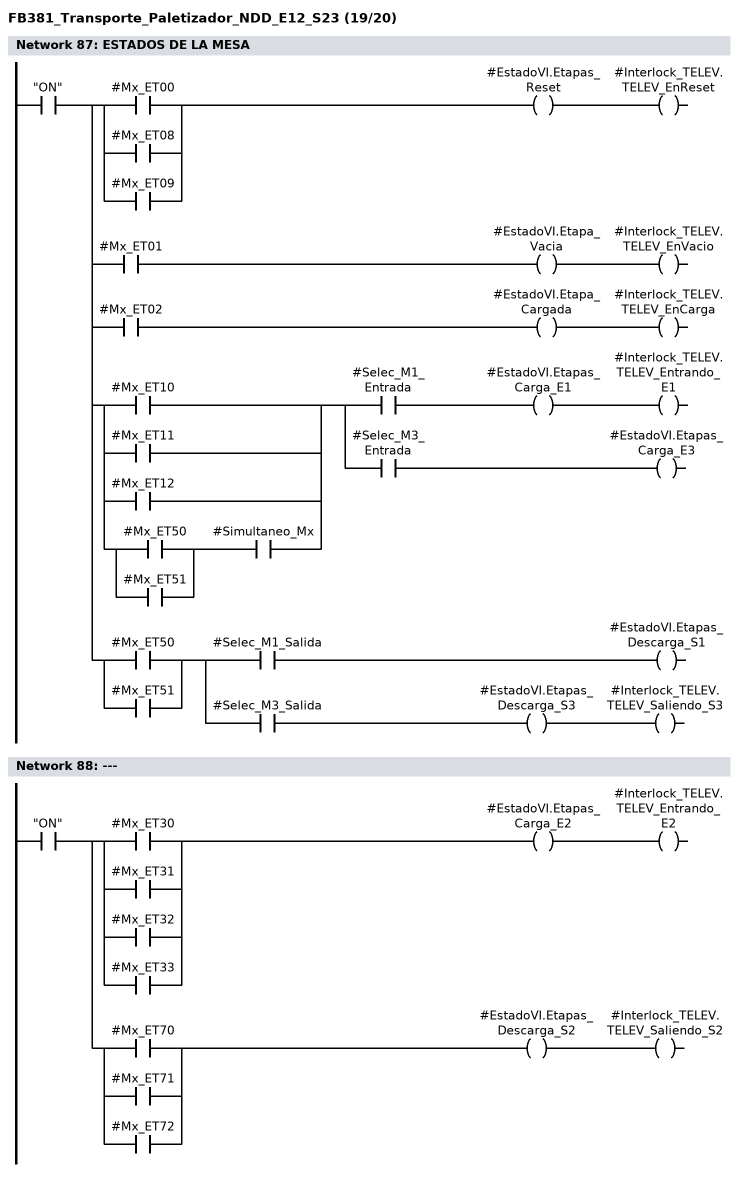
   RUNG wire#powerrail
      Contact( "ON" )
      wire#w1
      Contact( #Mx_ET00 )
      wire#w2
      Coil( #EstadoVI.Etapas_Reset )
      Coil( #Interlock_TELEV.TELEV_EnReset )
   END_RUNG
   RUNG wire#w1
      Contact( #Mx_ET08 )
   END_RUNG wire#w2
   RUNG wire#w1
      Contact( #Mx_ET09 )
   END_RUNG wire#w2
   RUNG wire#w1
      Contact( #Mx_ET01 )
      Coil( #EstadoVI.Etapa_Vacia )
      Coil( #Interlock_TELEV.TELEV_EnVacio )
   END_RUNG
   RUNG wire#w1
      Contact( #Mx_ET02 )
      Coil( #EstadoVI.Etapa_Cargada )
      Coil( #Interlock_TELEV.TELEV_EnCarga )
   END_RUNG
   RUNG wire#w1
      Contact( #Mx_ET10 )
      wire#w3
      Contact( #Selec_M1_Entrada )
      Coil( #EstadoVI.Etapas_Carga_E1 )
      Coil( #Interlock_TELEV.TELEV_Entrando_E1 )
   END_RUNG
   RUNG wire#w1
      Contact( #Mx_ET11 )
   END_RUNG wire#w3
   RUNG wire#w1
      Contact( #Mx_ET12 )
   END_RUNG wire#w3
   RUNG wire#w1
      Contact( #Mx_ET50 )
      wire#w4
      Contact( #Simultaneo_Mx )
   END_RUNG wire#w3
   RUNG wire#w1
      Contact( #Mx_ET51 )
   END_RUNG wire#w4
   RUNG wire#w3
      Contact( #Selec_M3_Entrada )
      Coil( #EstadoVI.Etapas_Carga_E3 )
   END_RUNG
   RUNG wire#w1
      Contact( #Mx_ET50 )
      wire#w5
      Contact( #Selec_M1_Salida )
      Coil( #EstadoVI.Etapas_Descarga_S1 )
   END_RUNG
   RUNG wire#w1
      Contact( #Mx_ET51 )
   END_RUNG wire#w5
   RUNG wire#w5
      Contact( #Selec_M3_Salida )
      Coil( #EstadoVI.Etapas_Descarga_S3 )
      Coil( #Interlock_TELEV.TELEV_Saliendo_S3 )
   END_RUNG
   // the same network as SCL:
   #EstadoVI.Etapas_Reset := "ON" AND (#Mx_ET00 OR #Mx_ET08 OR #Mx_ET09);
   #Interlock_TELEV.TELEV_EnReset := #EstadoVI.Etapas_Reset;
   #EstadoVI.Etapa_Vacia := "ON" AND #Mx_ET01;
   #Interlock_TELEV.TELEV_EnVacio := #EstadoVI.Etapa_Vacia;
   #EstadoVI.Etapa_Cargada := "ON" AND #Mx_ET02;
   #Interlock_TELEV.TELEV_EnCarga := #EstadoVI.Etapa_Cargada;
   #_w1 := "ON" AND (#Mx_ET10 OR #Mx_ET11 OR #Mx_ET12 OR ((#Mx_ET50 OR #Mx_ET51) AND #Simultaneo_Mx));
   #EstadoVI.Etapas_Carga_E1 := #_w1 AND #Selec_M1_Entrada;
   #Interlock_TELEV.TELEV_Entrando_E1 := #EstadoVI.Etapas_Carga_E1;
   #EstadoVI.Etapas_Carga_E3 := #_w1 AND #Selec_M3_Entrada;
   #_w2 := "ON" AND (#Mx_ET50 OR #Mx_ET51);
   #EstadoVI.Etapas_Descarga_S1 := #_w2 AND #Selec_M1_Salida;
   #EstadoVI.Etapas_Descarga_S3 := #_w2 AND #Selec_M3_Salida;
   #Interlock_TELEV.TELEV_Saliendo_S3 := #EstadoVI.Etapas_Descarga_S3;
END_REGION

REGION Network 88: ---
   RUNG wire#powerrail
      Contact( "ON" )
      wire#w1
      Contact( #Mx_ET30 )
      wire#w2
      Coil( #EstadoVI.Etapas_Carga_E2 )
      Coil( #Interlock_TELEV.TELEV_Entrando_E2 )
   END_RUNG
   RUNG wire#w1
      Contact( #Mx_ET31 )
   END_RUNG wire#w2
   RUNG wire#w1
      Contact( #Mx_ET32 )
   END_RUNG wire#w2
   RUNG wire#w1
      Contact( #Mx_ET33 )
   END_RUNG wire#w2
   RUNG wire#w1
      Contact( #Mx_ET70 )
      wire#w3
      Coil( #EstadoVI.Etapas_Descarga_S2 )
      Coil( #Interlock_TELEV.TELEV_Saliendo_S2 )
   END_RUNG
   RUNG wire#w1
      Contact( #Mx_ET71 )
   END_RUNG wire#w3
   RUNG wire#w1
      Contact( #Mx_ET72 )
   END_RUNG wire#w3
   // the same network as SCL:
   #EstadoVI.Etapas_Carga_E2 := "ON" AND (#Mx_ET30 OR #Mx_ET31 OR #Mx_ET32 OR #Mx_ET33);
   #Interlock_TELEV.TELEV_Entrando_E2 := #EstadoVI.Etapas_Carga_E2;
   #EstadoVI.Etapas_Descarga_S2 := "ON" AND (#Mx_ET70 OR #Mx_ET71 OR #Mx_ET72);
   #Interlock_TELEV.TELEV_Saliendo_S2 := #EstadoVI.Etapas_Descarga_S2;
END_REGION

REGION Network 89: ENTRADAS DE LA MESA
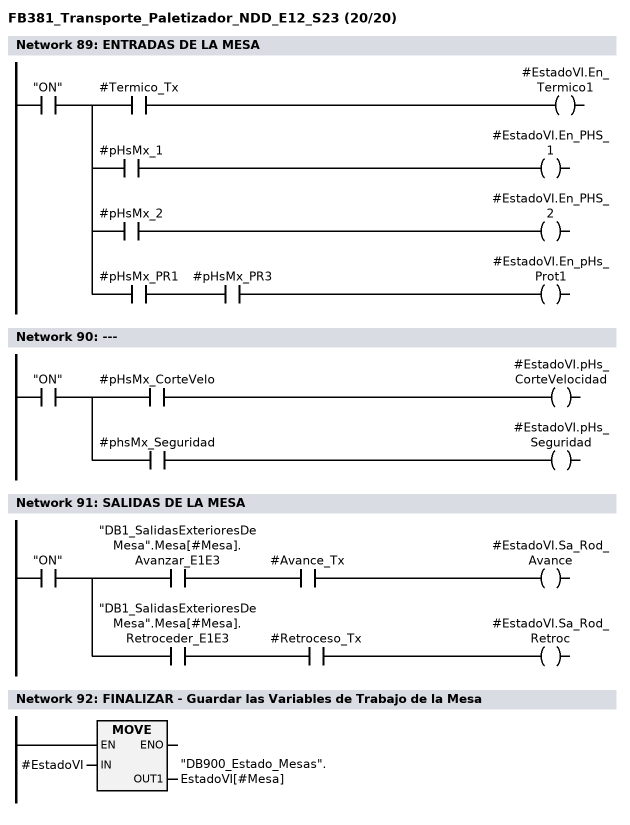
   RUNG wire#powerrail
      Contact( "ON" )
      wire#w1
      Contact( #Termico_Tx )
      Coil( #EstadoVI.En_Termico1 )
   END_RUNG
   RUNG wire#w1
      Contact( #pHsMx_1 )
      Coil( #EstadoVI.En_PHS_1 )
   END_RUNG
   RUNG wire#w1
      Contact( #pHsMx_2 )
      Coil( #EstadoVI.En_PHS_2 )
   END_RUNG
   RUNG wire#w1
      Contact( #pHsMx_PR1 )
      Contact( #pHsMx_PR3 )
      Coil( #EstadoVI.En_pHs_Prot1 )
   END_RUNG
   // the same network as SCL:
   #EstadoVI.En_Termico1 := "ON" AND #Termico_Tx;
   #EstadoVI.En_PHS_1 := "ON" AND #pHsMx_1;
   #EstadoVI.En_PHS_2 := "ON" AND #pHsMx_2;
   #EstadoVI.En_pHs_Prot1 := "ON" AND #pHsMx_PR1 AND #pHsMx_PR3;
END_REGION

REGION Network 90: ---
   RUNG wire#powerrail
      Contact( "ON" )
      wire#w1
      Contact( #pHsMx_CorteVelo )
      Coil( #EstadoVI.pHs_CorteVelocidad )
   END_RUNG
   RUNG wire#w1
      Contact( #phsMx_Seguridad )
      Coil( #EstadoVI.pHs_Seguridad )
   END_RUNG
   // the same network as SCL:
   #EstadoVI.pHs_CorteVelocidad := "ON" AND #pHsMx_CorteVelo;
   #EstadoVI.pHs_Seguridad := "ON" AND #phsMx_Seguridad;
END_REGION

REGION Network 91: SALIDAS DE LA MESA
   RUNG wire#powerrail
      Contact( "ON" )
      wire#w1
      Contact( "DB1_SalidasExterioresDeMesa".Mesa[#Mesa].Avanzar_E1E3 )
      Contact( #Avance_Tx )
      Coil( #EstadoVI.Sa_Rod_Avance )
   END_RUNG
   RUNG wire#w1
      Contact( "DB1_SalidasExterioresDeMesa".Mesa[#Mesa].Retroceder_E1E3 )
      Contact( #Retroceso_Tx )
      Coil( #EstadoVI.Sa_Rod_Retroc )
   END_RUNG
   // the same network as SCL:
   #EstadoVI.Sa_Rod_Avance := "ON" AND "DB1_SalidasExterioresDeMesa".Mesa[#Mesa].Avanzar_E1E3 AND #Avance_Tx;
   #EstadoVI.Sa_Rod_Retroc := "ON" AND "DB1_SalidasExterioresDeMesa".Mesa[#Mesa].Retroceder_E1E3 AND #Retroceso_Tx;
END_REGION

REGION Network 92: FINALIZAR - Guardar las Variables de Trabajo de la Mesa
   RUNG wire#powerrail
      Move(in := #EstadoVI, out1 => "DB900_Estado_Mesas".EstadoVI[#Mesa])
   END_RUNG
   // the same network as SCL:
   "DB900_Estado_Mesas".EstadoVI[#Mesa] := #EstadoVI;
END_REGION
END_FUNCTION_BLOCK
